METHOD ReadPropertyStatusFlags : HRESULT
VAR_INPUT
	stateFlags : REFERENCE TO ST_BA_StatusFlags;
END_VAR
VAR
	_flags : DWORD;
	_size : DINT := 2;
END_VAR
IF (ipObj <> 0) AND (__ISVALIDREF(stateFlags)) THEN
	ReadPropertyStatusFlags:=ReadProperty(E_BACnetPropIdentifier.PropStatusFlags, ADR(_flags), ADR(_size));
	
	IF (ReadPropertyStatusFlags = S_OK) THEN
		stateFlags.bInAlarm:= F_BACnet_IsBitFieldBitSet(_flags, E_BACnet_StatusFlags.eInAlarm);
		stateFlags.bFault:= F_BACnet_IsBitFieldBitSet(_flags, E_BACnet_StatusFlags.eFault);
		stateFlags.bOverridden:= F_BACnet_IsBitFieldBitSet(_flags, E_BACnet_StatusFlags.eOverridden);
		stateFlags.bOutOfService:= F_BACnet_IsBitFieldBitSet(_flags, E_BACnet_StatusFlags.eOutOfService);
	END_IF
ELSE
	ReadPropertyStatusFlags := E_FAIL;
END_IF
END_METHOD

METHOD ReadPropertyString : HRESULT
VAR_INPUT
	ePropID : E_BACnetPropIdentifier;
	value : REFERENCE TO T_MaxString;
END_VAR
VAR
	_size : UDINT := 255;
	_fbDecode : FB_BACnet_StringExtDecode;
END_VAR
IF (ipObj <> 0) AND (__ISVALIDREF(value)) THEN
	_size:=SIZEOF(BACnet_Globals.stADSBuffer);
	ReadPropertyString:=ReadProperty(ePropID, ADR(BACnet_Globals.stADSBuffer), ADR(_size));
	
	IF (ReadPropertyString = S_OK) THEN
		memset(ADR(value)+_size,0,1);
		_fbDecode(pChrStringExt:=ADR(BACnet_Globals.stADSBuffer), pOutString:=ADR(value), nOutSize:=_size);
		
		IF NOT _fbDecode.bValid THEN
			ReadPropertyString := E_FAIL;	
		END_IF
	END_IF
ELSE
	ReadPropertyString := E_FAIL;
END_IF
END_METHOD

METHOD ReadPropertyUDInt : HRESULT
VAR_INPUT
	ePropID : E_BACnetPropIdentifier;
	value : REFERENCE TO UDINT;
END_VAR
VAR
	_size : DINT := 4;
END_VAR
IF (ipObj <> 0) AND (__ISVALIDREF(value)) THEN
	ReadPropertyUDInt := ReadProperty(ePropID, ADR(value), ADR(_size));
ELSE
	ReadPropertyUDInt := E_FAIL;
END_IF
END_METHOD

METHOD ReadPropertyUnit : HRESULT
VAR CONSTANT
	ePropID : E_BACnetPropIdentifier := E_BACnetPropIdentifier.PropUnits;
END_VAR
VAR_INPUT
	value : REFERENCE TO E_BA_Unit;
END_VAR
VAR
	_size : DINT := 4;
END_VAR
IF (ipObj <> 0) AND (__ISVALIDREF(value)) THEN
	ReadPropertyUnit := ReadProperty(ePropID, ADR(value), ADR(_size));
ELSE
	ReadPropertyUnit := E_FAIL;
END_IF
END_METHOD

METHOD ReadPropertyWeeklySched : HRESULT
VAR_IN_OUT
	aWeek							: ARRAY[*, *] OF ST_BA_SchedEntry;
END_VAR
VAR_INPUT
	eDatatype						: E_BACnet_ValueChoice;
END_VAR
VAR			
	// General:
	nLenTmp							: UDINT;
	nLength							: DINT;
	
	_cbTmpSize						: UDINT;
	_cbTotalEntry					: UDINT;
	_cbTotalBuf						: UDINT;
	
	// Scheduler:
	_pDailySched					: POINTER TO ST_BACnet_DailySchedule;
	_pTimeValue						: POINTER TO ST_BACnet_TimeValueList;
	_pOldTimeValue					: POINTER TO ST_BACnet_TimeValueList;
	_nDayTmp						: DINT;
	_nDayEntryTmp					: DINT;
	_nDays							: UINT;
END_VAR
IF (ipObj = 0) THEN
	_hResult := E_FAIL;
	
ELSIF (eDataType = E_BACnet_ValueChoice.eNullValue) THEN
	iOwner.LogMsg.Show(ADSLOG_MSGTYPE_ERROR, 'RWS05', 'Invalid datatype!', TRUE);
	_hResult := E_FAIL;
ELSE
	nLength := SIZEOF(BACnet_Globals.aDefaultBuffer);
	_hResult := ReadProperty(E_BACnetPropIdentifier.PropWeeklySchedule, ADR(BACnet_Globals.aDefaultBuffer), ADR(nLength));
	
	IF (SUCCEEDED(_hResult)) THEN
		IF (nLength > 0) THEN
			// Clear content:
			_nDayTmp := F_BA_WeeklySchedSize(aWeek);
			MEMSET(aWeek, 0, TO_UDINT(F_BA_WeeklySchedSize(aWeek)));
			
			// Point to first data:
			_pDailySched := ADR(BACnet_Globals.aDefaultBuffer);
			_pTimeValue := ADR(_pDailySched^.stListEntry);
			_nDayEntryTmp := LOWER_BOUND(aWeek, 2);
			_nDayTmp := LOWER_BOUND(aWeek, 1);
			
			WHILE (_pTimeValue <> 0) AND SUCCEEDED(_hResult) DO
				(* check entry size of time value *)
				IF (_pTimeValue^.nEntrySize AND 16#7FFFFFFF) > 0 THEN
					(* check internal schedule buffer index *)
					IF (_nDayTmp > E_BA_Weekday.eSunday) THEN
						iOwner.LogMsg.Show(ADSLOG_MSGTYPE_ERROR, 'RWS23', 'Wrong day index!', TRUE);
						_hResult := E_FAIL;
					ELSE
						IF (_nDayEntryTmp <= TO_INT(BACnet_Globals.nDataField_MaxDayEntry)) THEN
							Sched_ReadEntry(eDatatype, _pTimeValue, ADR(aWeek[_nDayTmp, _nDayEntryTmp]));							
							_nDayEntryTmp := _nDayEntryTmp + 1;
						ELSE
							iOwner.LogMsg.Show(ADSLOG_MSGTYPE_WARN, 'RWS74', 'Max. count of entries reached!', TRUE);
						END_IF
	
						(* next time value entry *)
						(* check if next time value entry available *)
						IF (NOT Sched_SetNextTimeVal(_pDailySched, _pTimeValue, _cbTmpSize, _pOldTimeValue)) THEN
							(* update pointer each cycle (even if no day follows!) *)
							(* check for next day *)
							IF (NOT Sched_SetNextDay(_pDailySched, _cbTmpSize, _cbTotalBuf, _pOldTimeValue, _nDayTmp, _nDayEntryTmp, _pTimeValue)) THEN
								// Job done!
								EXIT;
							END_IF
						END_IF
					END_IF
	
				ELSE
					(* update pointer each cycle (even if no day follows!) *)
					(* No timevalue entry, check if next day element exists and pointer is plausible *)
					IF (Sched_SetNextDay(_pDailySched, _cbTmpSize, _cbTotalBuf, _pOldTimeValue, _nDayTmp, _nDayEntryTmp, _pTimeValue)) THEN
						
						// Check pointer:
						IF (_pDailySched + (_pDailySched^.nEntrySize AND 16#7FFFFFFF)) >= (ADR(BACnet_Globals.aDefaultBuffer) + SIZEOF(BACnet_Globals.aDefaultBuffer)) THEN
							iOwner.LogMsg.Show(ADSLOG_MSGTYPE_ERROR, 'RWS96', 'Insufficient buffer size!', TRUE);
							_hResult := E_FAIL;
						END_IF
					ELSE
						// Job done!
						EXIT;
					END_IF
				END_IF
				
				// Check bounds:
				IF (_nDayTmp > UPPER_BOUND(aWeek, 1)) OR (_nDayEntryTmp > UPPER_BOUND(aWeek, 2)) THEN
					EXIT;
				END_IF
			END_WHILE
		END_IF
	END_IF
END_IF

ReadPropertyWeeklySched := _hResult;
END_METHOD

METHOD INTERNAL GetSyncHandleMode : BOOL
VAR_INPUT
	eMode		: E_BA_FullSyncMode;
END_VAR
VAR_OUTPUT
	eResult		: E_BA_SyncMode;
END_VAR
CASE (eMode) OF
	eSync_FromSupplement:
		eResult := E_BA_SyncMode.eFromSupplement;
		
	eSync_ToSupplement,
	eFullSync_InitSupplement,
	eFullSync_InitPLC:
		eResult := E_BA_SyncMode.eToSupplement;
ELSE
	eResult := E_BA_SyncMode.eNone;
END_CASE

GetSyncHandleMode := (eResult <> E_BA_SyncMode.eNone);
END_METHOD

METHOD PRIVATE AddListElement : BOOL
VAR_INPUT
	ePropID				: E_BACnetPropIdentifier;
	nIndex				: DINT;
	nSize				: DINT;
	pValue				: PVOID;
END_VAR
VAR
	nListLen			: DINT;
	_size				: DINT := SIZEOF(DINT);
END_VAR
// Read current element count:
IF ipObj.SyncReadProperty(ePropID, ADR(nListLen), ADR(_size), 0) = S_OK THEN
	IF nListLen < nIndex THEN
		// Add new element to list:
		AddListElement := (ipObj.SyncWriteProperty(ePropID, pValue, nSize, 16#FFFFFFFE) = S_OK);
	ELSE
		AddListElement := TRUE;
	END_IF
END_IF
END_METHOD

METHOD PRIVATE ApplySyncHandler : BOOL
VAR
	_i		: E_BA_SyncMode;
END_VAR
ApplySyncHandler := TRUE;

// Apply requested sync handlers:
FOR _i := E_BA_SyncMode.eFromSupplement TO E_BA_SyncMode.eToSupplement DO
	IF (aReqSyncHandlers[_i] > 0) THEN
		IF (NOT SetPropertyCount(aReqSyncHandlers[_i], _i)) THEN
			ApplySyncHandler := FALSE;
		END_IF
	END_IF
END_FOR
END_METHOD

METHOD PRIVATE EvaluatePropSync
VAR_INPUT
	hResult		: HRESULT;
	eSyncMode	: E_BA_FullSyncMode;
	bCyclic		: BOOL := FALSE;
END_VAR
VAR
	_eMode		: E_BA_SyncMode	:= E_BA_SyncMode.eNone;
END_VAR
IF (SUCCEEDED(hResult)) THEN
	// Cyclic property synchronization:
	IF ((bCyclic) AND (eSyncMode > eSync_FromSupplement)) THEN
		nCycPropCnt := (nCycPropCnt+1);
	END_IF
	
	// Increment SyncHandlers:
	IF (GetSyncHandleMode(eSyncMode, eResult=>_eMode)) THEN
		aSyncHandlers[_eMode] := (aSyncHandlers[_eMode]+1);
	END_IF
END_IF
END_METHOD

METHOD RequestSyncHandlers : BOOL
VAR_INPUT
	nFromSupplement		: UDINT		:= 0;
	nToSupplement		: UDINT		:= 0;
END_VAR
aReqSyncHandlers[E_BA_SyncMode.eFromSupplement] := (aReqSyncHandlers[E_BA_SyncMode.eFromSupplement]+nFromSupplement);
aReqSyncHandlers[E_BA_SyncMode.eToSupplement] := (aReqSyncHandlers[E_BA_SyncMode.eToSupplement]+nToSupplement);
END_METHOD

METHOD RequestSyncHandlersEx : BOOL
VAR_INPUT
	eMode		: E_BA_FullSyncMode;
	nCount		: UDINT		:= 0;
END_VAR
VAR
	_eMode		: E_BA_SyncMode	:= E_BA_SyncMode.eNone;
END_VAR
IF (GetSyncHandleMode(eMode, eResult=>_eMode)) THEN
	aReqSyncHandlers[_eMode] := (aReqSyncHandlers[_eMode]+nCount);
	
	RequestSyncHandlersEx := TRUE;
END_IF
END_METHOD

METHOD SyncProperty : HRESULT
VAR_INPUT
	ePropID : E_BACnetPropIdentifier;
	nSize : UDINT;
	pValue : PVOID;
	bCOVTrig : POINTER TO BOOL := 0;
	eSyncMode : E_BA_FullSyncMode;
	bCyclic : BOOL := FALSE;
END_VAR
VAR
	nIndex : UDINT := 16#FFFFFFFF;
	_bCOV		: POINTER TO BYTE;
END_VAR
IF (ipObj <> 0) THEN
	SyncProperty := SEL(Error, ipObj.SyncPropertyData(ePropID, nSize, pValue, bCOVTrig, 0, nIndex, TO_UINT(eSyncMode)), E_FAIL);
	EvaluatePropSync(SyncProperty, eSyncMode, bCyclic);
	
	IF (SUCCEEDED(SyncProperty)) AND_THEN (bCOVTrig <> 0) THEN
		// Initialize COV indication:
		bCOVTrig^ := FALSE;
	END_IF
	
				
END_IF
END_METHOD

METHOD SyncPropertyCOV : BOOL
VAR_INPUT
	ePropertyID : E_BACnetPropIdentifier;
	bCOVTrig : POINTER TO BOOL;
END_VAR
VAR
	_hResult : HRESULT;
END_VAR
IF (ipObj <> 0) AND_THEN (bCOVTrig <> 0) THEN
	// Initialize COV indication:
	_hResult := SyncProperty(ePropertyID, 0, 0, bCOVTrig, eSync_FromSupplement, FALSE);
	IF (_hResult <> S_OK) THEN
		iOwner.LogMsg.Show2(ADSLOG_MSGTYPE_ERROR, 'SPCOV03', 'Initialize COV-Trigger of property "%d" failed (Error: 0x%x)!', F_INT(ePropertyID), F_DINT(_hResult), TRUE);
	ELSE
		// Initialize COV indication:
		bCOVTrig^ := FALSE;
		
		SyncPropertyCOV := TRUE;
	END_IF
END_IF
END_METHOD

METHOD SyncPropertyIdx : HRESULT
VAR_INPUT
	ePropID : E_BACnetPropIdentifier;
	nSize : UDINT;
	pValue : PVOID;
	nIndex : INT := -1;
	pData : PVOID := 0;
	eSyncMode : E_BA_FullSyncMode;
	bCyclic : BOOL := FALSE;
END_VAR
IF (ipObj <> 0) THEN
	SyncPropertyIdx := SEL(Error, ipObj.SyncPropertyData(ePropID, nSize, pValue, pData, 0, TO_UDINT(nIndex), TO_UINT(eSyncMode)), E_FAIL);
	EvaluatePropSync(_hResult, eSyncMode, bCyclic);
END_IF
END_METHOD

METHOD SyncPropertyList : BOOL
VAR_INPUT
	ePropID				: E_BACnetPropIdentifier;
	pList				: PVOID;
	nItemSize			: UDINT;
	nItemCount			: UDINT;
	eSyncMode			: E_BA_FullSyncMode;
	bValidate			: BOOL						:= FALSE;			// Check items contents and stops synchronization if an used items is found.
END_VAR
VAR
	_nTemp				: UDINT;
	_pValue				: PVOID;
END_VAR
IF (bValidate) THEN
	RemoveListElements(ePropID);
END_IF

IF (ipObj <> 0) AND_THEN (pList <> 0) AND (nItemSize > 0) AND (nItemCount > 0) THEN
	FOR _nTemp := 1 TO nItemCount DO
		_pValue := (pList + ((_nTemp-1) * nItemSize));
		
		IF (bValidate) AND_THEN (F_BA_ByteCmp(_pValue, nItemSize, 0) = 0) THEN
			// Synchronization of used items completed:
			EXIT;
		END_IF
	
		IF NOT AddListElement(ePropID, TO_DINT(_nTemp), SIZEOF(STRING), _pValue) THEN
			RETURN;
		ELSIF SyncPropertyIdx(ePropID, SIZEOF(STRING), _pValue, TO_INT(_nTemp), 0, eSyncMode, FALSE) <> S_OK THEN
			RETURN;
		END_IF
	END_FOR
	
	SyncPropertyList := TRUE;
END_IF
END_METHOD

METHOD SyncPropertyPvPrio : HRESULT
VAR_INPUT
	ePropID : E_BACnetPropIdentifier;
	nSize : UDINT;
	pValue : PVOID;
	bEnPriority : POINTER TO BOOL;
	ePriority : E_BACnet_Priority;
	pData : PVOID := 0;
	eSyncMode : E_BA_FullSyncMode;
	bCyclic : BOOL := FALSE;
END_VAR
IF (ipObj <> 0) THEN
	SyncPropertyPvPrio := SEL(Error, ipObj.SyncPropertyData(ePropID, nSize, pValue, pData, bEnPriority, TO_UDINT(ePriority), TO_UINT(eSyncMode)), E_FAIL);
	EvaluatePropSync(_hResult, eSyncMode, bCyclic);
END_IF
END_METHOD

METHOD WriteProperty : HRESULT
VAR_INPUT
	ePropID : E_BACnetPropIdentifier;
	pData : PVOID;
	nData : DINT;
END_VAR
IF (ipObj <> 0) THEN
	WriteProperty:=ipObj.SyncWriteProperty(TO_INT(ePropID), pData, nData, 16#FFFFFFFF);
	
	IF (WriteProperty <> S_OK) THEN
		iOwner.LogMsg.Show2(ADSLOG_MSGTYPE_ERROR, 'WP5', 'Writing property "%d" failed (Error "0x%x")!', F_INT(ePropID), F_DINT(WriteProperty), TRUE);
	END_IF
ELSE
	WriteProperty := E_FAIL;
END_IF
END_METHOD

METHOD WritePropertyBool : HRESULT
VAR_INPUT
	ePropID : E_BACnetPropIdentifier;
	bValue : BOOL;
END_VAR
IF (ipObj <> 0) THEN
	WritePropertyBool := WriteProperty(ePropID, ADR(bValue), SIZEOF(bValue));
ELSE
	WritePropertyBool := E_FAIL;
END_IF
END_METHOD

METHOD WritePropertyDateList : HRESULT
VAR_IN_OUT
	aDateList				: ARRAY[*] OF ST_BA_CalendarEntry;
END_VAR
VAR
	_i						: DINT;
	
	_stEntry				: POINTER TO ST_BACnet_CalendarEntry;
	_cbTotalBuf				: UDINT;
END_VAR
IF (ipObj = 0) THEN
	_hResult := E_FAIL;
ELSE
	_stEntry := ADR(BACnet_Globals.aDefaultBuffer);
	_cbTotalBuf := 0;
	
	FOR _i := LOWER_BOUND(aDateList, 1) TO UPPER_BOUND(aDateList, 1) DO
		IF (F_BACnet_ToDateListEntry(ADR(aDateList[_i]), stResult=>_stEntry^)) THEN		
			_stEntry := (_stEntry+SIZEOF(ST_BACnet_CalendarEntry));
			_cbTotalBuf := (_cbTotalBuf+SIZEOF(ST_BACnet_CalendarEntry));
		END_IF
	END_FOR
	
	// Write data:
	_hResult := WriteProperty(E_BACnetPropIdentifier.PropDateList, ADR(BACnet_Globals.aDefaultBuffer), TO_DINT(_cbTotalBuf));
END_IF	

WritePropertyDateList := _hResult;
END_METHOD

METHOD WritePropertyEventEnable : HRESULT
VAR_INPUT
	bToNormal : BOOL;
	bToFault : BOOL;
	bToOffNormal : BOOL;
END_VAR
VAR
	_flags : WORD := 16#0005;
END_VAR
IF (ipObj <> 0) THEN
	IF bToNormal THEN
		_flags:=_flags OR 16#2000;
	END_IF
	IF bToFault THEN
		_flags:=_flags OR 16#4000;
	END_IF
	IF bToOffNormal THEN
		_flags:=_flags OR 16#8000;
	END_IF

	WritePropertyEventEnable := WriteProperty(E_BACnetPropIdentifier.PropEventEnable, ADR(_flags), 2);
ELSE
	WritePropertyEventEnable := E_FAIL;
END_IF
END_METHOD

METHOD WritePropertyEventParameter : HRESULT
VAR_IN_OUT
	stEventParameter		: ST_BACnet_EventParameter;
END_VAR
VAR
	_cbTotalBuf				: UDINT;
END_VAR
IF (ipObj = 0) THEN
	_hResult := E_FAIL;
ELSE
	CASE stEventParameter.eEventType OF
		E_BACnet_EventType.eOutOfRange:
			stEventParameter.nArgSize := SIZEOF(ST_BACnet_EventOutOfRange);
		E_BACnet_EventType.eUnsignedRange:
			stEventParameter.nArgSize := SIZEOF(ST_BACnet_EventUnsignedRange);
		ELSE
			IF stEventParameter.nArgSize = 0 THEN
				WritePropertyEventParameter := E_FAIL;
				RETURN;
			END_IF
	END_CASE
	_cbTotalBuf := TO_UDINT(8 + stEventParameter.nArgSize);
	_hResult := WriteProperty(E_BACnetPropIdentifier.PropEventParameters, ADR(stEventParameter), TO_DINT(_cbTotalBuf));
END_IF	

WritePropertyEventParameter := _hResult;
END_METHOD

METHOD WritePropertyExceptionSched : HRESULT
VAR_IN_OUT
	aCalendar			: ARRAY[*] OF ST_BACnet_SchedCalendar;
	aException			: ARRAY[*] OF ST_BACnet_SchedException;
END_VAR
VAR_INPUT
	eDatatype			: E_BACnet_ValueChoice;
END_VAR
VAR
	_nEntry				: DINT;
	_nSchedEntry		: INT;
	_hResult			: HRESULT;
	_pDailySched		: POINTER TO ST_BACnet_SpecialEventList;
	_pDailySchedOld		: POINTER TO ST_BACnet_SpecialEventList;
	_cbTotalSize		: UDINT;
	_cbTmpSize			: UDINT;
	_calObjId 			: T_BACnet_ObjectIdentifier;
	_pTimeValue			: POINTER TO ST_BACnet_TimeValueList;
	_pOldTimeValue		: POINTER TO ST_BACnet_TimeValueList;
	
	// [Bug-Workaround]: Diese scheiss Firma 3S
	// CASE (aCalendar[_nEntry].aEntry[_nSchedEntry].eState) OF			// "...aEntry[_nTimeValue]" ist immer der Pointer auf "aEntry[1]" :(
	_pCalEntry			: POINTER TO ST_BA_SchedEntry;
	
	// [Bug-Workaround]: Diese scheiss Firma 3S
	// Sched_ReadEntry(eDatatype, _pTimeValue, aException[_nExcEntry].aEntry[_nTimeValue]);			// "...aEntry[_nTimeValue]" ist immer der Pointer auf "aEntry[1]" :(
	_pExceptEntry		: POINTER TO ST_BA_SchedEntry;
END_VAR
IF ipObj = 0 THEN
	_hResult := E_FAIL;
ELSE
	_pDailySched := ADR(BACnet_Globals.aDefaultBuffer);
	_pDailySchedOld := 0;
	_cbTotalSize := 0;
	
	FOR _nEntry := LOWER_BOUND(aCalendar, 1) TO UPPER_BOUND(aCalendar, 1) DO
		IF F_BACnet_IsObjIdentifierValid(aCalendar[_nEntry].tRefCalendarID) THEN
			MEMSET(ADR(_pDailySched^.stEvent), 0, SIZEOF(_pDailySched^.stEvent));
			_pDailySched^.nEntrySize := SIZEOF(_pDailySched^.stEvent);
			_pDailySched^.nRes := 0;
			_pDailySched^.stEvent.eEventChoice := E_BACnet_SpecialEventChoice.eCalendarReference;
			_pDailySched^.stEvent.nEventPriority := SEL(F_BACnet_IsPriorityValid(aCalendar[_nEntry].eEventPriority), 1, TO_UDINT(aCalendar[_nEntry].eEventPriority));
				
			IF  _pDailySchedOld <> 0 THEN
				_pDailySchedOld^.nEntrySize := _pDailySchedOld^.nEntrySize + 16#80000000;
			END_IF
			
			_calObjId := aCalendar[_nEntry].tRefCalendarID;
			MEMCPY(ADR(_pDailySched^.stEvent.eCalEntryChoice), ADR(_calObjId), SIZEOF(_calObjId));
			
			_pOldTimeValue := 0;
			_pTimeValue:= F_BACnet_EndOf(_pDailySched, SIZEOF(ST_BACnet_SpecialEventList));
			_pCalEntry := ADR(aCalendar[_nEntry].aEntry[1]);
			FOR _nSchedEntry:=1 TO BACnet_Param.nSched_EntryCount DO
				CASE (_pCalEntry^.eState) OF
					E_BA_SchedEntryState.eNull,
					E_BA_SchedEntryState.eValue:
						 _pTimeValue^.nEntrySize := 0;
						 _pTimeValue^.nRes := 0;
						 
						 // Set flag "next entry" to the previous element:
						IF (_nSchedEntry > 1) AND (_pOldTimeValue <> 0) THEN
							_pOldTimeValue^.nEntrySize := _pOldTimeValue^.nEntrySize + 16#80000000;
						END_IF
						
						Sched_WriteEntry(eDatatype, _pTimeValue, _pCalEntry); 
						
						_pDailySched^.nEntrySize := _pDailySched^.nEntrySize + F_BACnet_AlignedSize(_pTimeValue^.nEntrySize) + SIZEOF(_pTimeValue^.nEntrySize) + SIZEOF(_pTimeValue^.nRes);	
											
						_pOldTimeValue := _pTimeValue;
						_pTimeValue := _pTimeValue +  F_BACnet_AlignedSize(_pTimeValue^.nEntrySize AND 16#7FFFFFFF) + SIZEOF(_pTimeValue^.nEntrySize) + SIZEOF(_pTimeValue^.nRes);					 
				END_CASE
				_pCalEntry := (_pCalEntry+SIZEOF(ST_BA_SchedEntry));
			END_FOR
			IF _pOldTimeValue = 0 THEN // no TimeValue entry -> empty list
				_pDailySched^.nEntrySize := _pDailySched^.nEntrySize + SIZEOF(_pTimeValue^.nEntrySize) + SIZEOF(_pTimeValue^.nRes);
				_pTimeValue^.nEntrySize := 0;
				_pTimeValue^.nRes := 0;
			END_IF
		
			_cbTotalSize := _cbTotalSize + F_BACnet_AlignedSize(_pDailySched^.nEntrySize AND 16#7FFFFFFF) + SIZEOF(_pDailySched^.nEntrySize) + SIZEOF(_pDailySched^.nRes);	
			_pDailySchedOld := _pDailySched;
			_pDailySched := _pDailySched +  F_BACnet_AlignedSize(_pDailySched^.nEntrySize AND 16#7FFFFFFF) + SIZEOF(_pDailySched^.nEntrySize) + SIZEOF(_pDailySched^.nRes);					 		
		END_IF
	END_FOR
	
	FOR _nEntry := LOWER_BOUND(aException, 1) TO UPPER_BOUND(aException, 1) DO
		IF aException[_nEntry].eType <> E_BA_DateValChoice.Invalid THEN
			MEMSET(ADR(_pDailySched^.stEvent), 0, SIZEOF(_pDailySched^.stEvent));
			_pDailySched^.nEntrySize := SIZEOF(_pDailySched^.stEvent);
			_pDailySched^.nRes := 0;
			_pDailySched^.stEvent.eEventChoice := E_BACnet_SpecialEventChoice.eCalendarEntry;
			IF aException[_nEntry].nEventPriority > 0 AND aException[_nEntry].nEventPriority < 17 THEN
				_pDailySched^.stEvent.nEventPriority := aException[_nEntry].nEventPriority; 
			ELSE
				_pDailySched^.stEvent.nEventPriority := 1;
			END_IF
			IF _pDailySchedOld <> 0 THEN
				_pDailySchedOld^.nEntrySize := _pDailySchedOld^.nEntrySize + 16#80000000;
			END_IF
			
			_pDailySched^.stEvent.eCalEntryChoice := aException[_nEntry].eType-1;
			_pDailySched^.stEvent.uCalEntry := aException[_nEntry].uDate;
			
			_pOldTimeValue := 0;
			_pTimeValue:= F_BACnet_EndOf(_pDailySched, SIZEOF(ST_BACnet_SpecialEventList));
			_pExceptEntry := ADR(aException[_nEntry].aEntry[1]);
			FOR _nSchedEntry:=1 TO BACnet_Param.nSched_EntryCount DO
				CASE (_pExceptEntry^.eState) OF
					E_BA_SchedEntryState.eNull,
					E_BA_SchedEntryState.eValue:
						 _pTimeValue^.nEntrySize := 0;
						 _pTimeValue^.nRes := 0;
						 
						 // Set flag "next entry" to the previous element:
						IF (_nSchedEntry > 1) AND (_pOldTimeValue <> 0) THEN
							_pOldTimeValue^.nEntrySize := _pOldTimeValue^.nEntrySize + 16#80000000;
						END_IF
						
						Sched_WriteEntry(eDatatype, _pTimeValue, _pExceptEntry); 
						
						_pDailySched^.nEntrySize := _pDailySched^.nEntrySize + F_BACnet_AlignedSize(_pTimeValue^.nEntrySize) + SIZEOF(_pTimeValue^.nEntrySize) + SIZEOF(_pTimeValue^.nRes);	
											
						_pOldTimeValue := _pTimeValue;
						_pTimeValue := _pTimeValue +  F_BACnet_AlignedSize(_pTimeValue^.nEntrySize AND 16#7FFFFFFF) + SIZEOF(_pTimeValue^.nEntrySize) + SIZEOF(_pTimeValue^.nRes);					 
				END_CASE
				_pExceptEntry := (_pExceptEntry+SIZEOF(ST_BA_SchedEntry));
			END_FOR
			IF _pOldTimeValue = 0 THEN // no TimeValue entry -> empty list
				_pDailySched^.nEntrySize := _pDailySched^.nEntrySize + SIZEOF(_pTimeValue^.nEntrySize) + SIZEOF(_pTimeValue^.nRes);
				_pTimeValue^.nEntrySize := 0;
				_pTimeValue^.nRes := 0;
			END_IF
						
			_cbTotalSize := _cbTotalSize + F_BACnet_AlignedSize(_pDailySched^.nEntrySize AND 16#7FFFFFFF) + SIZEOF(_pDailySched^.nEntrySize) + SIZEOF(_pDailySched^.nRes);	
			_pDailySchedOld := _pDailySched;
			_pDailySched := _pDailySched +  F_BACnet_AlignedSize(_pDailySched^.nEntrySize AND 16#7FFFFFFF) + SIZEOF(_pDailySched^.nEntrySize) + SIZEOF(_pDailySched^.nRes);					 
		END_IF
	END_FOR
	
	IF (_cbTotalSize = 0) THEN
		// Indicate empty exception property:
		_cbTotalSize := 8;
		MEMSET(ADR(BACnet_Globals.aDefaultBuffer), 0, _cbTotalSize);
	END_IF
	
	// Write data:
	_hResult := WriteProperty(E_BACnetPropIdentifier.PropExceptionSchedule, ADR(BACnet_Globals.aDefaultBuffer), TO_DINT(_cbTotalSize));
END_IF

IF (F_BACnet_FilterErrCode(_hResult) = TO_DINT(E_AdsErr.DEVICE_ACCESSDENIED)) THEN
	// Fallback to old (valid) property value:
	ReadPropertyExceptionSched(aCalendar, aException, eDataType);
END_IF

WritePropertyExceptionSched := _hResult;
END_METHOD

METHOD WritePropertyLimitEnable : HRESULT
VAR_INPUT
	bLowLimitEnable : BOOL;
	bHighLimitEnable : BOOL;
END_VAR
VAR
	_flags : WORD := 16#0006;
END_VAR
IF (ipObj <> 0) THEN
	IF bLowLimitEnable THEN
		_flags:=_flags OR 16#8000;
	END_IF
	IF bHighLimitEnable THEN
		_flags:=_flags OR 16#4000;
	END_IF

	WritePropertyLimitEnable := WriteProperty(E_BACnetPropIdentifier.PropLimitEnable, ADR(_flags), 2);
ELSE
	WritePropertyLimitEnable := E_FAIL;
END_IF
END_METHOD

METHOD WritePropertyLogBuffer : HRESULT
VAR_IN_OUT
	aLogBuffer						: ARRAY [*] OF ST_BA_TrendEntry;
END_VAR
IF (ipObj = 0) THEN
	_hResult := E_FAIL;
ELSE
	_hResult := S_OK;
	// ...
	
END_IF	

WritePropertyLogBuffer := _hResult;
END_METHOD

METHOD WritePropertyNotifyType : HRESULT
VAR CONSTANT
	ePropID : E_BACnetPropIdentifier := E_BACnetPropIdentifier.PropNotifyType;
END_VAR
VAR_INPUT
	value : E_BACnet_NotifyType;
END_VAR
IF (ipObj <> 0) THEN
	WritePropertyNotifyType := WriteProperty(ePropID, ADR(value), SIZEOF(value));
ELSE
	WritePropertyNotifyType := E_FAIL;
END_IF
END_METHOD

METHOD WritePropertyNull : HRESULT
VAR_INPUT
	ePropID : E_BACnetPropIdentifier;
	prio : BYTE := 0;
END_VAR
IF (ipObj <> 0) THEN
	WritePropertyNull := ipObj.SyncWriteProperty(TO_INT(ePropID), 0, 0, prio);
	
	IF (WritePropertyNull <> S_OK) THEN
		F_BA_LogMessage2(ADSLOG_MSGTYPE_ERROR, 'WPN5', 'Writing property "%d" failed (Error "0x%x")!', F_INT(ePropID), F_DINT(WritePropertyNull));
	END_IF
ELSE
	WritePropertyNull := E_FAIL;
END_IF
END_METHOD

METHOD WritePropertyReal : HRESULT
VAR_INPUT
	ePropID : E_BACnetPropIdentifier;
	fValue : REAL;
END_VAR
IF (ipObj <> 0) THEN
	WritePropertyReal := WriteProperty(ePropID, ADR(fValue), SIZEOF(fValue));
ELSE
	WritePropertyReal := E_FAIL;
END_IF
END_METHOD

METHOD WritePropertyRealPrio : HRESULT
VAR_INPUT
	ePropID : E_BACnetPropIdentifier;
	fValue : REAL;
	prio : BYTE := 0;
END_VAR
IF (ipObj <> 0) THEN
	WritePropertyRealPrio := ipObj.SyncWriteProperty(TO_INT(ePropID), ADR(fValue), SIZEOF(fValue), prio);
	
	IF (WritePropertyRealPrio <> S_OK) THEN
		F_BA_LogMessage2(ADSLOG_MSGTYPE_ERROR, 'WPRP5', 'Writing property "%d" failed (Error "0x%x")!', F_INT(ePropID), F_DINT(WritePropertyRealPrio));
	END_IF
ELSE
	WritePropertyRealPrio := E_FAIL;
END_IF
END_METHOD

METHOD WritePropertyRecipientList : HRESULT
VAR_IN_OUT
	aRecipientList			: ARRAY[*] OF ST_BACnet_Destination;
END_VAR
// [Bugworkaround]
// > _stUnused" has to be static, otherwise its memory can be initialized incorrectly by PLC :(
VAR_STAT
	_nLowerBound			: DINT;
	_nCount					: DINT;
	_stUnused				: ST_BACnet_Destination;
END_VAR
_hResult := E_FAIL;

IF (ipObj <> 0) THEN
	_nLowerBound := LOWER_BOUND(aRecipientList, 1);
	_nCount := F_BA_GetUsedEntryCount(aRecipientList, _nLowerBound, UPPER_BOUND(aRecipientList, 1), _stUnused);
	
	IF (_nCount > 0) THEN
		_hResult := WriteProperty(E_BACnetPropIdentifier.PropRecipientList, aRecipientList, SIZEOF(ST_BACnet_Destination) * (_nLowerBound + _nCount - 1));
	ELSE
		IF RemoveArrayElements(E_BACnetPropIdentifier.PropRecipientList) THEN
			_hResult := S_OK;
		END_IF
	END_IF
END_IF

IF (F_BACnet_FilterErrCode(_hResult) = TO_DINT(E_AdsErr.DEVICE_ACCESSDENIED)) THEN
	// Fallback to old (valid) property value:
	ReadPropertyRecipientList(aRecipientList);
END_IF

WritePropertyRecipientList := _hResult;
END_METHOD

METHOD WritePropertyReference : HRESULT
VAR_INPUT
	eProperty			: E_BACnetPropIdentifier;
END_VAR
VAR_IN_OUT
	stReference			: ST_BACnet_ObjectPropertyReference;
END_VAR
VAR
	_pEntry				: ST_BACnet_DeviceObjectPropertyReference;
END_VAR
IF (ipObj <> 0) THEN
	IF (stReference.iObject = 0) THEN
		// Set referred object to NULL.
	ELSE
		_pEntry.stValidFields.bPropertyIdentifier := TRUE;
		_pEntry.stValidFields.bObjectId := TRUE;
		_pEntry.tObjId := stReference.iObject.ObjectID;
		_pEntry.ePropIdentifier := stReference.ePropertyId;
	END_IF
	
	WritePropertyReference := WriteProperty(eProperty, ADR(_pEntry), SIZEOF(_pEntry));
ELSE
	WritePropertyReference := E_FAIL;
END_IF
END_METHOD

METHOD WritePropertyReferenceList : HRESULT
VAR_INPUT
	eProperty			: E_BACnetPropIdentifier;
END_VAR
VAR_IN_OUT
	aReferences 		: ARRAY[*] OF ST_BACnet_ObjectPropertyReference;
END_VAR
VAR
	_pEntry				: POINTER TO ST_BACnet_DeviceObjectPropertyReference;
	_i 					: DINT;
	_nSize				: DINT;
END_VAR
IF (ipObj <> 0) THEN
	_pEntry := ADR(BACnet_Globals.aDefaultBuffer);

	FOR _i:= LOWER_BOUND(aReferences, 1) TO UPPER_BOUND(aReferences, 1) DO
		IF (aReferences[_i].iObject <> 0) THEN
			MEMSET(_pEntry, 0, SIZEOF(ST_BACnet_DeviceObjectPropertyReference));
			
			_pEntry^.stValidFields.bPropertyIdentifier := TRUE;
			_pEntry^.stValidFields.bObjectId := TRUE;
			_pEntry^.tObjId := aReferences[_i].iObject.ObjectID;
			_pEntry^.ePropIdentifier := aReferences[_i].ePropertyId;
			
			_nSize := _nSize + SIZEOF(ST_BACnet_DeviceObjectPropertyReference);
			_pEntry := F_BACnet_EndOf(_pEntry, SIZEOF(ST_BACnet_DeviceObjectPropertyReference));
		END_IF
	END_FOR
	WritePropertyReferenceList := WriteProperty(eProperty, ADR(BACnet_Globals.aDefaultBuffer),_nSize);
ELSE
	WritePropertyReferenceList := E_FAIL;
END_IF
END_METHOD

METHOD WritePropertyReferenceList1x : HRESULT
VAR_INPUT
	eProperty			: E_BACnetPropIdentifier;
END_VAR
VAR_IN_OUT
	stReference			: ST_BACnet_ObjectPropertyReference;
END_VAR
VAR
	_aRefArray 			: POINTER TO ARRAY[1 .. 1] OF ST_BACnet_ObjectPropertyReference;
END_VAR
IF (ipObj <> 0) THEN
	_aRefArray := ADR(stReference);
	WritePropertyReferenceList1x := WritePropertyReferenceList(eProperty, _aRefArray^);
ELSE
	WritePropertyReferenceList1x := E_FAIL;
END_IF
END_METHOD

METHOD WritePropertyString : HRESULT
VAR_INPUT
	ePropID : E_BACnetPropIdentifier;
	value : T_MaxString;
END_VAR
VAR
	_nResult : UDINT;
END_VAR
IF (ipObj <> 0) THEN
	IF (F_BACnet_EncodeUTF8(
		pString		:= ADR(value),
		nString	:= TO_UDINT(LEN(value)),
		pResult		:= ADR(BACnet_Globals.stADSBuffer),
		nResult	:= SIZEOF(BACnet_Globals.stADSBuffer),
		nResultLen	:= _nResult) <> 0)
			THEN
				WritePropertyString := WriteProperty(ePropID, ADR(BACnet_Globals.stADSBuffer), TO_UINT(_nResult));
	END_IF
END_IF
END_METHOD

METHOD WritePropertyStringIdx : HRESULT
VAR_INPUT
	ePropID : E_BACnetPropIdentifier;
	str : STRING;
	idx : BYTE;
END_VAR
VAR
	_nResult : UDINT;
END_VAR
IF (ipObj <> 0) THEN
	IF (F_BACnet_EncodeUTF8(
		pString		:= ADR(str),
		nString	:= TO_UDINT(LEN(str)),
		pResult		:= ADR(BACnet_Globals.stADSBuffer),
		nResult	:= SIZEOF(BACnet_Globals.stADSBuffer),
		nResultLen	:= _nResult) <> 0)
			THEN
			WritePropertyStringIdx := ipObj.SyncWriteProperty(TO_INT(ePropID), ADR(BACnet_Globals.stADSBuffer),  TO_UINT(F_BACnet_AlignedSize(_nResult)), idx);
			
			IF (WritePropertyStringIdx <> S_OK) THEN
				F_BA_LogMessage2(ADSLOG_MSGTYPE_ERROR, 'WPSI512', 'Writing property "%d" failed (Error "0x%x")!', F_INT(ePropID), F_DINT(WritePropertyStringIdx));
			END_IF
	END_IF
END_IF
END_METHOD

METHOD WritePropertyUDInt : HRESULT
VAR_INPUT
	ePropID : E_BACnetPropIdentifier;
	nValue : UDINT;
END_VAR
IF (ipObj <> 0) THEN
	WritePropertyUDInt := WriteProperty(ePropID, ADR(nValue), SIZEOF(nValue));
ELSE
	WritePropertyUDInt := E_FAIL;
END_IF
END_METHOD

METHOD WritePropertyUInt : HRESULT
VAR_INPUT
	ePropID : E_BACnetPropIdentifier;
	nValue : UINT;
END_VAR
IF (ipObj <> 0) THEN
	WritePropertyUInt := WriteProperty(ePropID, ADR(nValue), SIZEOF(nValue));
ELSE
	WritePropertyUInt := E_FAIL;
END_IF
END_METHOD

METHOD WritePropertyUnit : HRESULT
VAR CONSTANT
	ePropID : E_BACnetPropIdentifier := E_BACnetPropIdentifier.PropUnits;
END_VAR
VAR_INPUT
	eValue : E_BA_Unit;
END_VAR
IF (ipObj <> 0) THEN
	WritePropertyUnit := WriteProperty(ePropID, ADR(eValue), SIZEOF(eValue));
ELSE
	WritePropertyUnit := E_FAIL;
END_IF
END_METHOD

METHOD WritePropertyValue : HRESULT
VAR_INPUT
	eProperty : E_BACnetPropIdentifier;
	xValue : ANY;
END_VAR
VAR
	_eValueChoice : E_BACnet_ValueChoice;
END_VAR
CASE (xValue.TypeClass) OF
	__SYSTEM.TYPE_CLASS.TYPE_REAL:
		_eValueChoice := E_BACnet_ValueChoice.eRealValue;
	__SYSTEM.TYPE_CLASS.TYPE_UDINT:
		_eValueChoice := E_BACnet_ValueChoice.eUnsignedValue;
	__SYSTEM.TYPE_CLASS.TYPE_BOOL:
		_eValueChoice := E_BACnet_ValueChoice.eBoolValue;
	__SYSTEM.TYPE_CLASS.TYPE_ENUM:
		_eValueChoice := E_BACnet_ValueChoice.eEnumerationValue;
ELSE
	iOwner.LogMsg.Show1(ADSLOG_MSGTYPE_ERROR, 'WPV30', 'Unimplemented datatype! (Type class "%d")', F_DWORD(xValue.TypeClass), TRUE);
	RETURN;
END_CASE

WritePropertyValue := WritePropertyValueEx(eProperty, _eValueChoice, xValue.diSize, xValue.pValue);
END_METHOD

METHOD WritePropertyValueEx : HRESULT
VAR_INPUT
	eProperty : E_BACnetPropIdentifier;
	eValueChoice : E_BACnet_ValueChoice;
	nSize : DINT;
	pValue : PVOID;
END_VAR
VAR
	_stData : ST_BACnet_ValueList;
	_nSize : DWORD;
END_VAR
IF (bReady) AND (nSize > 0) AND (pValue <> 0) THEN
	IF (eValueChoice = E_BACnet_ValueChoice.eEnumerationValue) THEN
		_nSize := SIZEOF(ST_BACnet_ValueList);	
		_stData.nEntrySize := TO_DWORD(SIZEOF(ST_BACnet_Value));
		_stData.listEntry.eValueChoice := eValueChoice;
		_stData.listEntry.nSize := SIZEOF(ST_BACnet_EnumerationValueType);
		_stData.listEntry.stValue.choice := E_BACnet_EnumerationValueChoice.eBinaryPV;
		_stData.listEntry.stValue.enumValue := 0;
		
		MEMCPY(ADR(_stData.listEntry.stValue.enumValue), pValue, TO_UDINT(nSize)); 
	ELSE		
		_nSize := ((SIZEOF(ST_BACnet_ValueList) - SIZEOF(ST_BACnet_EnumerationValueType)) + TO_DWORD(nSize));
		
		_stData.nEntrySize := TO_DWORD((SIZEOF(ST_BACnet_Value) - SIZEOF(ST_BACnet_EnumerationValueType) + nSize));
		_stData.listEntry.eValueChoice := eValueChoice;
		_stData.listEntry.nSize := TO_DWORD(nSize);
		
		MEMCPY(ADR(_stData.listEntry.stValue), pValue, TO_UDINT(nSize)); 
	END_IF
	
	WritePropertyValueEx := WriteProperty(eProperty, ADR(_stData), TO_DINT(F_BACnet_AlignedSize(_nSize)));
				
	IF (S_OK <> WritePropertyValueEx) THEN
		iOwner.LogMsg.Show1(ADSLOG_MSGTYPE_ERROR, 'WPVE12', 'Writing value of property "%d" failed!', F_INT(eProperty), TRUE);
	END_IF
END_IF
END_METHOD

METHOD WritePropertyWeeklySched : HRESULT
VAR_IN_OUT
	aWeek					: ARRAY[*, *] OF ST_BA_SchedEntry;
END_VAR
VAR_INPUT
	eValueChoice			: E_BACnet_ValueChoice;
END_VAR
VAR
	_cbTmpSize				: UDINT;
	_cbTotalEntry			: UDINT;
	_cbTotalBuf				: UDINT;
	_pDailySched			: POINTER TO ST_BACnet_DailySchedule;
	_pTimeValue				: POINTER TO ST_BACnet_TimeValueList;
	_pOldTimeValue			: POINTER TO ST_BACnet_TimeValueList;
	_nDay					: DINT;
	_nDayEntry				: DINT;
	_nDays					: UINT;
END_VAR
IF (ipObj = 0) THEN
	_hResult := E_FAIL;
ELSE
	// Point to first data:
	_pDailySched := ADR(BACnet_Globals.aDefaultBuffer);
	_cbTotalBuf := 0;
	_nDay := LOWER_BOUND(aWeek, 1);
	_hResult := S_OK;
	
	WHILE SUCCEEDED(_hResult) DO
		// Set timevalue pointer:
		_pTimeValue := ADR(_pDailySched^.stListEntry);
		_pTimeValue^.nEntrySize := 0;
		_pTimeValue^.nRes := 0;
		_cbTotalEntry := 0;
		_pOldTimeValue := 0;
		
		FOR _nDayEntry := LOWER_BOUND(aWeek, 2) TO UPPER_BOUND(aWeek, 2) DO			
			CASE (aWeek[_nDay, _nDayEntry].eState) OF
				E_BA_SchedEntryState.eNull,
				E_BA_SchedEntryState.eValue:
					// Set flag "next entry" to the previous element:
					IF (_nDayEntry > 1) AND (_pOldTimeValue <> 0) THEN
						_pOldTimeValue^.nEntrySize := _pOldTimeValue^.nEntrySize + 16#80000000;
					END_IF
					
					Sched_WriteEntry(eValueChoice, _pTimeValue, ADR(aWeek[_nDay, _nDayEntry])); 
					
					// Update time value pointer:
					Sched_SetNextTimeVal(_pDailySched, _pTimeValue, _cbTmpSize, _pOldTimeValue);
					
					// ...and add to total entry size counter:
					_cbTotalEntry := _cbTotalEntry + _cbTmpSize;
			END_CASE
		END_FOR
		
		// Caclulate day-entry size:
		_pDailySched^.nEntrySize := MAX(_cbTotalEntry, SIZEOF(_pDailySched^.stListEntry.nEntrySize) + SIZEOF(_pDailySched^.stListEntry.nRes));
		
		// Next day?
		IF (_nDay < UPPER_BOUND(aWeek, 1)) THEN
			_pDailySched^.nEntrySize := _pDailySched^.nEntrySize + 16#80000000;
		END_IF
		
		// Update pointer each cycle (even if no day follows!):
		IF NOT Sched_SetNextDay(_pDailySched, _cbTmpSize, _cbTotalBuf, _pOldTimeValue, _nDay, _nDayEntry, _pTimeValue) THEN
			EXIT;
		END_IF
	END_WHILE
	
	// Write data:
	_hResult := WriteProperty(E_BACnetPropIdentifier.PropWeeklySchedule, ADR(BACnet_Globals.aDefaultBuffer), TO_DINT(_cbTotalBuf));
END_IF	
	
IF (F_BACnet_FilterErrCode(_hResult) = TO_DINT(E_AdsErr.DEVICE_ACCESSDENIED)) THEN
	// Fallback to old (valid) property value:
	ReadPropertyWeeklySched(aWeek, eValueChoice);
END_IF

WritePropertyWeeklySched := _hResult;
END_METHOD

END_FUNCTION_BLOCK

// POUs/Helper/F_BACnet_GetObjId
FUNCTION F_BACnet_GetObjId : T_BACnet_ObjectIdentifier
VAR_INPUT
	eObjectType		: E_BACnetObjType;
	nObjectInstance	: UDINT;
END_VAR
VAR
END_VAR

F_BACnet_GetObjId := F_BACnet_GetObjInstance(nObjectInstance) + SHL(INT_TO_UDINT(eObjectType), 22);

END_FUNCTION

// POUs/Helper/F_BACnet_GetObjInstance
FUNCTION F_BACnet_GetObjInstance : UDINT
VAR_INPUT
	nObjectId : DWORD;
END_VAR
VAR
END_VAR

F_BACnet_GetObjInstance := nObjectId AND BACnet_Globals.nBACnetInstId_Auto;

END_FUNCTION

// POUs/Helper/F_BACnet_GetObjType
FUNCTION F_BACnet_GetObjType : E_BACnetObjType
VAR_INPUT
	nObjectId : DWORD;
END_VAR
VAR
END_VAR

F_BACnet_GetObjType := TO_INT(SHR((nObjectId AND 16#FFC00000), 22));

END_FUNCTION

// POUs/Local/Objects/FB_BACnet_View
// Structured View Object
{attribute 'enable_dynamic_creation'}
FUNCTION_BLOCK FB_BACnet_View EXTENDS FB_BACnet_Object IMPLEMENTS I_BACnet_View
VAR_INPUT CONSTANT
	{attribute 'parameterCategory':='General'}
	eNodeType : E_BACnet_NodeType := E_BACnet_NodeType.eOrganizational;
END_VAR
VAR
	{region 'Linked Object-List'}
		{attribute 'hide'}
		iFirstChild				: I_BACnet_Object;
		{attribute 'hide'}
		iLastChild				: I_BACnet_Object;
		{attribute 'no_copy'}
		nChildCount				: DINT;
	{endregion}
END_VAR
VAR_STAT
	{region 'Internal'}
		// (BETA) ... Following symbols should be made non-static / thread safe!
		{attribute 'hide'}
		iThisView				: I_BACnet_View;
	{endregion}
END_VAR

SUPER^();

// Unused - Implemented for compatibility reason!
{attribute 'hide'}
METHOD Close
iFirstChild := 0;
iLastChild := 0;
nChildCount := 0;

SUPER^.Close();
END_METHOD

{attribute 'hide'}
METHOD AddObject : BOOL
VAR_INPUT
	iObject			: I_BACnet_Object;
END_VAR
VAR_OUTPUT
	nResultIndex	: DINT;
END_VAR
IF (iObject <> 0) THEN
	iThisView := THIS^;
	
	IF (iObject.Parent = 0) THEN
		fbLogMsg.Show(ADSLOG_MSGTYPE_ERROR, 'AO05', 'No parent defined in child-object!', FALSE);
		
	ELSIF (iObject.Parent <> iThisView) THEN
		fbLogMsg.Show(ADSLOG_MSGTYPE_ERROR, 'AO07', 'Child already assigned to another parent!', FALSE);
		
	ELSE
		IF (FindObject(iObject, nResultIndex)) THEN
			// Child already assigned.
		ELSE
			// Register 'iObject' as a new child in the linked list:
			nResultIndex := nChildCount;
			
			IF (nChildCount = 0) THEN
				iFirstChild := iObject;
			ELSE
				iLastChild.NextSibling := iObject;
				iObject.PrevSibling := iLastChild;
			END_IF
			iLastChild := iObject;
			nChildCount := (nChildCount + 1);
			
			IF (bReady) THEN
				// Register child object:
				View_AddSubordinate(iObject);
			END_IF
		END_IF
		
		AddObject := TRUE;
	END_IF
END_IF
END_METHOD

{attribute 'hide'}
METHOD RemoveObject : BOOL
VAR_INPUT
	iObject			: I_BACnet_Object;
END_VAR
VAR
	_nTemp			: DINT;
	_fbObj			: POINTER TO FB_BACnet_Object;
END_VAR
IF (iObject <> 0) THEN
	iThisView := THIS^;
	
	IF (iObject.Parent = iThisView) AND (FindObject(iObject, _nTemp) <> 0) THEN
		IF (__QUERYPOINTER(iObject, _fbObj)) THEN
			// Remove object from linked object list of current instance:
			_fbObj^.RemoveFromLinkedObjList(iFirstChild, iLastChild);
			nChildCount := (nChildCount-1);
			
			RemoveObject := TRUE;
		END_IF
	END_IF
	
	iObject.Parent := 0;
	iObject.PrevSibling := 0;
	iObject.NextSibling := 0;
END_IF
END_METHOD

METHOD PROTECTED OnObjectStateChanged
VAR
	_iObj			: I_BACnet_Object;
END_VAR
SUPER^.OnObjectStateChanged();

CASE (tState) OF
	TCOM_STATE.TCOM_STATE_PREOP:
		// SyncHandler:
		RequestSyncHandlers(0, 1);
		
	TCOM_STATE.TCOM_STATE_SAFEOP:
		;

	TCOM_STATE.TCOM_STATE_OP:
		SyncProperty(E_BACnetPropIdentifier.PropNodeType, SIZEOF(eNodeType), ADR(eNodeType), 0, eFullSync_InitPLC, FALSE);

		// Add so far registered child objects to subordinate list:
		_iObj := iFirstChild;
		WHILE (_iObj <> 0) DO
			View_AddSubordinate(_iObj);
			_iObj := _iObj.NextSibling;
		END_WHILE

END_CASE
END_METHOD

METHOD FB_init : BOOL
VAR_INPUT
	bInitRetains : BOOL; // if TRUE, the retain variables are initialized (warm start / cold start)
	bInCopyCode : BOOL;  // if TRUE, the instance afterwards gets moved into the copy code (online change)
END_VAR
eObjectType := E_BACnetObjType.ObjStructuredView;
END_METHOD

METHOD FindObject : BOOL
VAR_INPUT
	iObject			: I_BACnet_Object;
END_VAR
VAR_IN_OUT
	nResultIndex	: DINT;
END_VAR
VAR
	_iObj			: I_BACnet_Object;
END_VAR
FindObject := FALSE;

IF (iObject <> 0) THEN
	_iObj := iFirstChild;
	nResultIndex := 0;
	
	WHILE (_iObj <> 0) DO
		IF (_iObj = iObject) THEN
			FindObject := TRUE;
			RETURN;
		ELSE
			nResultIndex := (nResultIndex + 1);
			_iObj := _iObj.NextSibling;
		END_IF
	END_WHILE
END_IF
END_METHOD

END_FUNCTION_BLOCK

// POUs/Helper/[internal]/F_BACnet_AlignedSize
{attribute 'hide'} // [Workaround] Not hidden when lib is included
FUNCTION INTERNAL F_BACnet_AlignedSize : DWORD
VAR_INPUT
	n	: DWORD;
END_VAR
VAR
END_VAR

F_BACnet_AlignedSize := (4*(((n)+3)/4));

END_FUNCTION

// POUs/Helper/[internal]/F_BACnet_SetBitFieldBit
{attribute 'hide'} // [Workaround] Not hidden when lib is included
FUNCTION INTERNAL F_BACnet_SetBitFieldBit : DWORD
VAR_INPUT
	ptrData		:	POINTER TO DWORD;
	bitNbr			:	INT;
END_VAR
VAR
END_VAR

ptrData^ := ptrData^ OR (SHR(DWORD#16#00008000, F_BACnet_BitFieldBit(bitNbr)));
F_BACnet_SetBitFieldBit := ptrData^;

END_FUNCTION

// POUs/Helper/[internal]/F_BACnet_BitFieldBit
{attribute 'hide'} // [Workaround] Not hidden when lib is included
FUNCTION INTERNAL F_BACnet_BitFieldBit : WORD
VAR_INPUT
	bitNbr	:	INT;
END_VAR
VAR
END_VAR

F_BACnet_BitFieldBit := to_word((bitNbr/8) * 8 + (bitNbr MOD 8));

END_FUNCTION

// POUs/Helper/[internal]/String/F_BACnet_EncodeUTF8
{attribute 'hide'} // [Workaround] Not hidden when lib is included
FUNCTION INTERNAL F_BACnet_EncodeUTF8 : UDINT (* actually byte length of the result utf-8 string (maybe longer than cbResult; means overflow) *)
VAR_INPUT
	pString		: POINTER TO BYTE; (* pointer to Win1252 string beginning *)
	nString	: UDINT; (* byte size of string (use SIZEOF - don't use LEN) *)
	pResult		: POINTER TO BYTE; (* pointer to result UTF-8 data area *)
	nResult	: UDINT; (* byte size of result (use SIZEOF - don't use LEN) *)
END_VAR

VAR
	pBy			: POINTER TO BYTE;
	pByArr		: POINTER TO ARRAY[0..3] OF BYTE;
	nCoded		: UINT;
	bOverflow	: BOOL;
END_VAR
(*All VAR_IN_OUT variables have been moved to the end of the declaration due to compatibility reasons*)
VAR_IN_OUT
	nResultLen	: UDINT; (* final resulting string length (<= nResult) *)
END_VAR

pBy			:= pString;
pByArr		:= pResult;
bOverflow	:= FALSE;
F_BACnet_EncodeUTF8 := 0;
nResultLen	:= 0;
(* loop over pString *)
WHILE pBy < (pString + nString) DO
	IF (pBy^ = 0) THEN EXIT; END_IF
	IF bOverflow OR (F_BACnet_EncodeUTF8 + 3 > nResult) THEN
		nCoded := F_BACnet_Win1252ToUtf8(nW1252:=pBy^, pUtf8:=pByArr, bEval:=TRUE);
		IF (NOT bOverflow) AND (F_BACnet_EncodeUTF8 + nCoded <= nResult) THEN
			nCoded := F_BACnet_Win1252ToUtf8(nW1252:=pBy^, pUtf8:=pByArr, bEval:=FALSE);
		ELSE
			bOverflow := TRUE;
		END_IF
	ELSE
		nCoded := F_BACnet_Win1252ToUtf8(nW1252:=pBy^, pUtf8:=pByArr, bEval:=FALSE);
	END_IF
	IF (NOT bOverflow) THEN
		pByArr := pByArr + UINT_TO_UDINT(nCoded);
		nResultLen := F_BACnet_EncodeUTF8 + nCoded;
	END_IF
	F_BACnet_EncodeUTF8 := F_BACnet_EncodeUTF8 + nCoded;
	pBy := pBy + 1;
END_WHILE
(* add zero termination if needed *)
IF (nResultLen < nResult) THEN
	pByArr^[0] := 16#00;
END_IF

END_FUNCTION

// POUs/Helper/[internal]/String/F_BACnet_Win1252ToUtf8
{attribute 'hide'} // [Workaround] Not hidden when lib is included
FUNCTION INTERNAL F_BACnet_Win1252ToUtf8 : UINT(0..3)
VAR_INPUT
	nW1252	: BYTE; (* Win1252 character *)
	pUtf8	: POINTER TO ARRAY[0..2] OF BYTE; (* pointer to target character buffer (utf-8) *)
	bEval	: BOOL; (* TRUE = only evaluate expected coding size (0..3 byte) - but don't write data *)
END_VAR
VAR
	pWord	: POINTER TO ARRAY[0..1] OF BYTE;
	wUCS2	: WORD;
END_VAR
VAR CONSTANT
	cRepl	: BYTE := 16#5F;
END_VAR

(*
	Windows-Codepages
874		Thai
932		Japanisch
936		Vereinfachtes Chinesisch
949		Koreanisch
950		Traditionelles Chinesisch
1250	Mitteleuropäisch
1251	Kyrillisch
1252	Westeuropäisch
1253	Griechisch
1254	Türkisch
1255	Hebräisch
1256	Arabisch
1257	Baltisch
1258	Vietnamesisch
*)
(* check pointer *)
IF (pUtf8 = 0) THEN
	(* null pointer *)
	F_BACnet_Win1252ToUtf8 := 0;
ELSIF (nW1252 <= 16#7F) THEN
	(* basic latin - 1 byte *)
	IF (NOT bEval) THEN
		pUtf8^[0] := nW1252;
	END_IF
	F_BACnet_Win1252ToUtf8 := 1;
ELSE
	(* convert to UCS-2 first *)
	wUCS2 := F_BACnet_Win1252ToUCS2(nW1252:=nW1252, bBE:=FALSE);
	pWord := ADR(wUCS2);
	(* convert used ranges *)
	IF (wUCS2 >= 16#80 AND wUCS2 <= 16#BF) THEN
		(* latin-1 supplement *)
		IF (NOT bEval) THEN
			pUtf8^[0] := 16#C2;
			pUtf8^[1] := pWord^[0];
		END_IF
		F_BACnet_Win1252ToUtf8 := 2;
	ELSIF (wUCS2 >= 16#C0 AND wUCS2 <= 16#FF) THEN
		(* latin-1 supplement *)
		IF (NOT bEval) THEN
			pUtf8^[0] := 16#C3;
			pUtf8^[1] := pWord^[0] - 16#40;
		END_IF
		F_BACnet_Win1252ToUtf8 := 2;
	ELSIF (wUCS2 >= 16#140 AND wUCS2 <= 16#17F) THEN
		(* latin extended A *)
		IF (NOT bEval) THEN
			pUtf8^[0] := 16#C5;
			pUtf8^[1] := pWord^[0] + 16#40;
		END_IF
		F_BACnet_Win1252ToUtf8 := 2;
	ELSIF (wUCS2 >= 16#20A0 AND wUCS2 <= 16#20BF) THEN
		(* currency symbols *)
		IF (NOT bEval) THEN
			pUtf8^[0] := 16#E2;
			pUtf8^[1] := 16#82;
			pUtf8^[2] := pWord^[0];
		END_IF
		F_BACnet_Win1252ToUtf8 := 3;
	ELSE
		(* unsupported *)
		IF (NOT bEval) THEN
			pUtf8^[0] := cRepl;
		END_IF
		F_BACnet_Win1252ToUtf8 := 1;
	END_IF
END_IF

END_FUNCTION

// POUs/Helper/[internal]/String/F_BACnet_Win1252ToUCS2
{attribute 'hide'} // [Workaround] Not hidden when lib is included
FUNCTION INTERNAL F_BACnet_Win1252ToUCS2 : WORD
VAR_INPUT
	nW1252 : BYTE;
	bBE	: BOOL; (* byte-order big endian = TRUE *)
END_VAR
VAR
	pArr : POINTER TO ARRAY[0..1] OF BYTE;
	nBuf : BYTE;
	wUCS2: WORD;
END_VAR

(*
	Windows-Codepages
874		Thai
932		Japanisch
936		Vereinfachtes Chinesisch
949		Koreanisch
950		Traditionelles Chinesisch
1250	Mitteleuropäisch
1251	Kyrillisch
1252	Westeuropäisch
1253	Griechisch
1254	Türkisch
1255	Hebräisch
1256	Arabisch
1257	Baltisch
1258	Vietnamesisch
*)
CASE nW1252 OF
	16#9F: wUCS2 := 16#178;
	16#9C: wUCS2 := 16#153;
	16#8C: wUCS2 := 16#152;
	16#9E: wUCS2 := 16#17E;
	16#8E: wUCS2 := 16#17D;
	16#9A: wUCS2 := 16#161;
	16#8A: wUCS2 := 16#160;
	16#80: wUCS2 := 16#20AC;
	ELSE
	wUCS2 := nW1252;
END_CASE
IF bBE THEN
	pArr := ADR(wUCS2);
	nBuf := pArr^[0];
	pArr^[0] := pArr^[1];
	pArr^[1] := nBuf;
END_IF
F_BACnet_Win1252ToUCS2 := wUCS2;

END_FUNCTION

// POUs/Helper/[internal]/F_BACnet_FilterErrCode
FUNCTION F_BACnet_FilterErrCode : HRESULT
VAR_INPUT
	hResult		: HRESULT;
END_VAR

F_BACnet_FilterErrCode := TO_UINT(hResult) AND 16#FFF;

END_FUNCTION

// POUs/Helper/[internal]/F_BACnet_IsBitFieldBitSet
{attribute 'hide'} // [Workaround] Not hidden when lib is included
FUNCTION INTERNAL F_BACnet_IsBitFieldBitSet : BOOL
VAR_INPUT
	data	:	DWORD;
	bitNbr		:	INT;
END_VAR
VAR
END_VAR

F_BACnet_IsBitFieldBitSet:= (data AND (SHR(DWORD#16#00008000,F_BACnet_BitFieldBit(bitNbr)))) > 0;

END_FUNCTION

// POUs/Helper/[internal]/Scheduler/F_BA_CalendarSchedSize
{attribute 'hide'}
FUNCTION F_BA_CalendarSchedSize : DINT
VAR_IN_OUT
	aCalendar			: ARRAY[*] OF ST_BACnet_SchedCalendar;
END_VAR

F_BA_CalendarSchedSize := (UPPER_BOUND(aCalendar, 1) - LOWER_BOUND(aCalendar, 1) + 1) * SIZEOF(ST_BACnet_SchedCalendar);

END_FUNCTION

// POUs/Helper/[internal]/Scheduler/F_BA_ExceptionSchedSize
{attribute 'hide'}
FUNCTION F_BA_ExceptionSchedSize : DINT
VAR_IN_OUT
	aException			: ARRAY[*] OF ST_BACnet_SchedException;
END_VAR

F_BA_ExceptionSchedSize := (UPPER_BOUND(aException, 1) - LOWER_BOUND(aException, 1) + 1) * SIZEOF(ST_BACnet_SchedException);

END_FUNCTION

// POUs/Helper/[internal]/F_BACnet_EndOf
{attribute 'hide'} // [Workaround] Not hidden when lib is included
FUNCTION INTERNAL F_BACnet_EndOf : POINTER TO BYTE
VAR_INPUT
	 pPtr : POINTER TO BYTE;
	 nSize : DWORD;
END_VAR
VAR
END_VAR

F_BACnet_EndOf:=pPtr+nSize;

END_FUNCTION

// POUs/Helper/[internal]/F_BACnet_NextListElem
{attribute 'hide'} // [Workaround] Not hidden when lib is included
FUNCTION INTERNAL F_BACnet_NextListElem : POINTER TO BYTE
VAR_INPUT
	 pPtr : POINTER TO BYTE;
	 nSize : DWORD;
END_VAR
VAR
END_VAR

IF nSize < 16#80000000 THEN
	F_BACnet_NextListElem:=0;
	RETURN;
END_IF
F_BACnet_NextListElem:=pPtr+F_BACnet_AlignedSize(nSize AND 16#7FFFFFFF)+8;

END_FUNCTION

// POUs/Helper/String/FB_BACnet_StringExtDecode
FUNCTION_BLOCK FB_BACnet_StringExtDecode (* convert UTF-8/UCS2/UCS4/ISO8859-1 to Windows-1252 *)
VAR_INPUT
	pChrStringExt	: POINTER TO ST_BACnet_CharacterStringExt; (* BACnet character string data structure (header and string) *)
	pOutString		: POINTER TO T_MaxString; (* pointer to result buffer (Windows-1252 encoded) *)
	nOutSize		: UDINT; (* byte size *)
END_VAR
VAR_OUTPUT
	bValid			: BOOL; (* Decoding successfull *)
	bOverflow		: BOOL; (* String length overflow (source string too long) *)
	bUnsupported	: BOOL; (* Souce encoding is unsupported (use ReadProp function and decode manually instead) *)
	nLength			: UDINT; (* out character length *)
	eSrcEncoding	: E_BACnet_StringEncodingTypes; (* input encoding *)
END_VAR
VAR
	pText 			: POINTER TO BYTE;
	pByte			: POINTER TO BYTE;
END_VAR

(* preset valid to FALSE *)
bValid := FALSE;
bOverflow := FALSE;
bUnsupported := FALSE;
(* check pointer *)
IF (pChrStringExt = 0) OR (pOutString = 0) THEN
	nLength := 0;
(* check input size *)
ELSIF (nOutSize = 0) THEN
	(* NULL string *)
	bValid := TRUE;
	pOutString^ := '';
	nLength := 0;
	eSrcEncoding := E_BACnet_StringEncodingTypes.eAnsiUtf8;
ELSE
	(* string data available *)
	IF (pChrStringExt^.cookie = 0) THEN
		(* new character string type *)
		nLength			:= UDINT_TO_UINT(pChrStringExt^.strLen);
		eSrcEncoding	:= UDINT_TO_INT(pChrStringExt^.encoding);
		pText			:= ADR(pChrStringExt^.aData);
	ELSE
		(* ASCII/UTF-8 string *)
		nLength			:= F_BACnet_ChrStrExtLen(pChrStringExt^);
		eSrcEncoding	:= E_BACnet_StringEncodingTypes.eAnsiUtf8;
		pText			:= pChrStringExt;
	END_IF

	(* check size *)
	IF (nLength = 0) THEN
		(* no data *)
		bValid := TRUE;
		pOutString^ := '';
	ELSIF (nLength <= nOutSize) THEN
		(* copy to output buffer first *)
		MEMMOVE(destAddr:= pOutString, srcAddr:= pText, n:= nLength);

		(* decode and copy *)
		CASE eSrcEncoding OF

			E_BACnet_StringEncodingTypes.eAnsiUtf8:
				bValid := TRUE;
				nLength := UDINT_TO_UINT(F_BACnet_DecodeUTF8(pOutString, nLength));

			E_BACnet_StringEncodingTypes.eUCS2:
				bValid := TRUE;
				nLength := UDINT_TO_UINT(F_BACnet_DecodeUCS2(pOutString, nLength));

			E_BACnet_StringEncodingTypes.eUCS4:
				bValid := TRUE;
				nLength := UDINT_TO_UINT(F_BACnet_DecodeUCS4(pOutString, nLength));

			E_BACnet_StringEncodingTypes.eISO8859:
				bValid := TRUE;
				(* check if string termination is already part of string *)
				pByte := pOutString + nLength - 1;
				IF (pByte^ = 16#00) THEN
					(* termination already part of string *)
					nLength := nLength - 1;
				ELSE
					(* add string termination *)
					pByte := pOutString + nLength;
					pByte^ := 16#00;
				END_IF

			ELSE
				bUnsupported := TRUE;

		END_CASE
	ELSE
		(* text too long *)
		nLength := 0;
		pOutString^ := '';
		bOverflow := TRUE;
	END_IF
END_IF

END_FUNCTION_BLOCK

// POUs/Helper/[internal]/String/F_BACnet_ChrStrExtLen
{attribute 'hide'} // [Workaround] Not hidden when lib is included
FUNCTION INTERNAL F_BACnet_ChrStrExtLen : UDINT
VAR
	pByte	: POINTER TO BYTE;
	nLen	: UDINT;
END_VAR
(*All VAR_IN_OUT variables have been moved to the end of the declaration due to compatibility reasons*)
VAR_IN_OUT
	stCharStringExt	: ST_BACnet_CharacterStringExt;
END_VAR

pByte := ADR(stCharStringExt);
nLen := SIZEOF(stCharStringExt);
(* check the string type *)
IF (nLen > 4 AND stCharStringExt.cookie = 0) THEN
	(* character string ext. *)
	IF (stCharStringExt.strLen <= SIZEOF(stCharStringExt.aData)) THEN
		(* plausible string length given *)
		F_BACnet_ChrStrExtLen := stCharStringExt.strLen;
		RETURN;
	END_IF
	(* use sizeof, because string length isn't plausible *)
	nLen := SIZEOF(stCharStringExt.aData);
	(* re-adjust pointer *)
	pByte := ADR(stCharStringExt.aData);
END_IF
(* scan zero termination *)
F_BACnet_ChrStrExtLen := 0;
WHILE ((pByte^ <> 0) AND (F_BACnet_ChrStrExtLen < nLen)) DO
	pByte := pByte + 1;
	F_BACnet_ChrStrExtLen := F_BACnet_ChrStrExtLen + 1;
END_WHILE

END_FUNCTION

// POUs/Helper/[internal]/String/F_BACnet_DecodeUTF8
{attribute 'hide'} // [Workaround] Not hidden when lib is included
FUNCTION INTERNAL F_BACnet_DecodeUTF8 : UDINT (* result is the new character length of the string *)
VAR_INPUT
	pString		: POINTER TO BYTE; (* pointer to UTF-8 string beginning *)
	nString	: UDINT; (* byte size of string (use SIZEOF - don't use LEN) *)
END_VAR
VAR
	i			: UDINT;
	pResult		: POINTER TO BYTE;
	pBy			: POINTER TO BYTE;
	pByArr		: POINTER TO ARRAY[0..3] OF BYTE;
END_VAR

pResult	:= pString;
pBy		:= pString;
FOR i := 0 TO nString-1 DO
	pByArr := pBy;
	IF (pByArr^[0] AND 16#F0) = 16#C0 THEN
		IF (pByArr^[1] AND 16#80) = 16#80 THEN
			pResult^ := F_BACnet_Utf8ToWin1252(pByArr, 2);
			pBy := pBy + 2;
		END_IF
	ELSIF (pByArr^[0] AND 16#F0) = 16#E0 THEN
		IF (pByArr^[1] AND 16#80) = 16#80 THEN
			IF (pByArr^[2] AND 16#80) = 16#80 THEN
				pResult^ := F_BACnet_Utf8ToWin1252(pByArr, 3);
				pBy := pBy + 3;
			END_IF
		END_IF
	ELSIF (pByArr^[0] AND 16#F0) = 16#F0 THEN
		IF (pByArr^[1] AND 16#80) = 16#80 THEN
			IF (pByArr^[2] AND 16#80) = 16#80 THEN
				IF (pByArr^[3] AND 16#80) = 16#80 THEN
					pResult^ := F_BACnet_Utf8ToWin1252(pByArr, 4);
					pBy := pBy + 4;
				END_IF
			END_IF
		END_IF
	ELSE
		(* ASCII character *)
		pResult^ := pBy^;
		pBy := pBy + 1;
	END_IF
	(* end-of-string by character *)
	IF (pResult^ = 16#00) THEN
		EXIT;
	END_IF
	(* next character *)
	pResult := pResult + 1;
	(* end-of-string by length *)
	IF (pBy >= (pString + nString)) THEN
		EXIT;
	END_IF
END_FOR
pResult^ := 16#00;
F_BACnet_DecodeUTF8 := pResult - pString;

END_FUNCTION

// POUs/Helper/[internal]/String/F_BACnet_Utf8ToWin1252
{attribute 'hide'} // [Workaround] Not hidden when lib is included
FUNCTION INTERNAL F_BACnet_Utf8ToWin1252 : BYTE
VAR_INPUT
	pUtf8	: POINTER TO BYTE;
	nUtf8	: UDINT; (* byte size of UTF8 character (1...6) *)
END_VAR
VAR
	pArr		: POINTER TO ARRAY[0..5] OF BYTE;
	pWord		: POINTER TO ARRAY[0..1] OF BYTE;
	wUCS2		: WORD;
END_VAR
VAR CONSTANT
	cRepl	: BYTE := 16#5F;
END_VAR

(*
	Windows-Codepages
874		Thai
932		Japanisch
936		Vereinfachtes Chinesisch
949		Koreanisch
950		Traditionelles Chinesisch
1250	Mitteleuropäisch
1251	Kyrillisch
1252	Westeuropäisch
1253	Griechisch
1254	Türkisch
1255	Hebräisch
1256	Arabisch
1257	Baltisch
1258	Vietnamesisch
*)
(* first step - convert to UCS2 *)
pArr := pUtf8;
IF (pArr^[0] <= 16#7F) THEN
	(* basic latin *)
	F_BACnet_Utf8ToWin1252 := pArr^[0];
	RETURN;
ELSIF (nUtf8 >= 2) THEN
	pWord := ADR(wUCS2);
	IF (pArr^[0] = 16#C2) THEN
		(* latin-1 supplement *)
		wUCS2 := pArr^[1];
	ELSIF (pArr^[0] = 16#C3) AND (pArr^[1] <= 16#BF) THEN
		(* latin-1 supplement *)
		wUCS2 := pArr^[1] + 16#40;
	ELSIF (pArr^[0] = 16#C4) AND (pArr^[1] >= 16#80) THEN
		(* latin extended-A *)
		pWord^[1] := 16#01;
		pWord^[0] := pArr^[1] - 16#80;
	ELSIF (pArr^[0] = 16#C5) AND (pArr^[1] >= 16#80) THEN
		(* latin extended-A *)
		pWord^[1] := 16#01;
		pWord^[0] := pArr^[1] - 16#40;
	ELSIF (pArr^[0] = 16#C6) AND (pArr^[1] >= 16#80) THEN
		(* latin extended-B *)
		pWord^[1] := 16#01;
		pWord^[0] := pArr^[1];
	ELSIF (pArr^[0] = 16#C7) AND (pArr^[1] <= 16#BF) THEN
		(* latin extended-B *)
		pWord^[1] := 16#01;
		pWord^[0] := pArr^[1] + 16#40;
	ELSIF (nUtf8 >= 3) THEN
		IF (pArr^[0] = 16#E2) AND (pArr^[1] = 16#82) THEN
			(* currency symbols *)
			pWord^[1] := 16#20;
			pWord^[0] := pArr^[2];
		ELSE
			(* unsupported *)
			F_BACnet_Utf8ToWin1252 := cRepl;
			RETURN;
		END_IF
	ELSE
		(* unsupported *)
		F_BACnet_Utf8ToWin1252 := cRepl;
		RETURN;
	END_IF
	(* convert UCS2 to Windows-1252 *)
	F_BACnet_Utf8ToWin1252 := F_BACnet_UCS2ToWin1252(pWord, FALSE);
	RETURN;
END_IF
(* unsupported *)
F_BACnet_Utf8ToWin1252 := cRepl;

END_FUNCTION

// POUs/Helper/[internal]/String/F_BACnet_UCS2ToWin1252
{attribute 'hide'} // [Workaround] Not hidden when lib is included
FUNCTION INTERNAL F_BACnet_UCS2ToWin1252 : BYTE
VAR_INPUT
	pUCS2 :	POINTER TO WORD;
	bBE	: BOOL; (* byte-order big endian = TRUE *)
END_VAR
VAR
	pArr : POINTER TO ARRAY[0..1] OF BYTE;
	wUCS2: WORD;
END_VAR
VAR CONSTANT
	cRepl	: BYTE := 16#5F;
END_VAR

(*
	Windows-Codepages
874		Thai
932		Japanisch
936		Vereinfachtes Chinesisch
949		Koreanisch
950		Traditionelles Chinesisch
1250	Mitteleuropäisch
1251	Kyrillisch
1252	Westeuropäisch
1253	Griechisch
1254	Türkisch
1255	Hebräisch
1256	Arabisch
1257	Baltisch
1258	Vietnamesisch
*)
pArr := pUCS2;
IF bBE THEN
	wUCS2 := (pArr^[0] * 16#0100) + pArr^[1];
ELSE
	wUCS2 := pUCS2^;
END_IF
CASE wUCS2 OF
	16#178: 	F_BACnet_UCS2ToWin1252 := 16#9F;
	16#153: 	F_BACnet_UCS2ToWin1252 := 16#9C;
	16#152: 	F_BACnet_UCS2ToWin1252 := 16#8C;
	16#17E: 	F_BACnet_UCS2ToWin1252 := 16#9E;
	16#17D: 	F_BACnet_UCS2ToWin1252 := 16#8E;
	16#161: 	F_BACnet_UCS2ToWin1252 := 16#9A;
	16#160: 	F_BACnet_UCS2ToWin1252 := 16#8A;
	16#20AC: 	F_BACnet_UCS2ToWin1252 := 16#80;
	ELSE
		IF wUCS2 <= 16#FF THEN
			F_BACnet_UCS2ToWin1252 := WORD_TO_BYTE(wUCS2);
		ELSE
			F_BACnet_UCS2ToWin1252 := cRepl;
		END_IF
END_CASE

END_FUNCTION

// POUs/Helper/[internal]/String/F_BACnet_DecodeUCS2
{attribute 'hide'} // [Workaround] Not hidden when lib is included
FUNCTION INTERNAL F_BACnet_DecodeUCS2 : UDINT (* result is the new character length of the string *)
VAR_INPUT
	pString		: POINTER TO WORD; (* pointer to UCS2 string beginning *)
	nString	: UDINT; (* byte size of string (use SIZEOF - don't use LEN) *)
END_VAR
VAR
	i		: UDINT;
	pResult	: POINTER TO BYTE;
	pBy		: POINTER TO WORD;
END_VAR

pResult	:= pString;
pBy		:= pString;
FOR i := 0 TO nString-1 DO
	pResult^ := F_BACnet_UCS2ToWin1252(pBy, TRUE);
	pBy := pBy + 2;
	(* end-of-string by character *)
	IF (pResult^ = 16#00) THEN
		EXIT;
	END_IF
	(* next character *)
	pResult := pResult + 1;
	(* end-of-string by length *)
	IF (pBy >= (pString + nString)) THEN
		EXIT;
	END_IF
END_FOR
pResult^ := 16#00;
F_BACnet_DecodeUCS2 := pResult - pString;

END_FUNCTION

// POUs/Helper/[internal]/String/F_BACnet_DecodeUCS4
{attribute 'hide'} // [Workaround] Not hidden when lib is included
FUNCTION INTERNAL F_BACnet_DecodeUCS4 : UDINT (* result is the new character length of the string *)
VAR_INPUT
	pString		: POINTER TO DWORD; (* pointer to UCS4 string beginning *)
	nString	: UDINT; (* byte size of string (use SIZEOF - don't use LEN) *)
END_VAR
VAR
	i		: UDINT;
	pResult	: POINTER TO BYTE;
	pBy		: POINTER TO WORD;
END_VAR

pResult	:= pString;
pBy		:= pString;
FOR i := 0 TO nString-1 DO
	(* byte order big endian *)
	pResult^ := F_BACnet_UCS2ToWin1252(pBy+2, TRUE);
	pBy := pBy + 4;
	(* end-of-string by character *)
	IF (pResult^ = 16#00) THEN
		EXIT;
	END_IF
	(* next character *)
	pResult := pResult + 1;
	(* end-of-string by length *)
	IF (pBy >= (pString + nString)) THEN
		EXIT;
	END_IF
END_FOR
pResult^ := 16#00;
F_BACnet_DecodeUCS4 := pResult - pString;

END_FUNCTION

// POUs/Helper/[internal]/Validation-Functions/F_BACnet_IsObjIdentifierValid
{attribute 'hide'} // [Workaround] Not hidden when lib is included
FUNCTION INTERNAL F_BACnet_IsObjIdentifierValid : BOOL
VAR_INPUT
	tIdentifier		: T_BACnet_ObjectIdentifier;
END_VAR

F_BACnet_IsObjIdentifierValid := ((tIdentifier <> 0) AND_THEN (tIdentifier <> BACnet_Globals.nBACnetObjId_None));

END_FUNCTION

// POUs/Helper/[internal]/Validation-Functions/F_BACnet_IsPriorityValid
{attribute 'hide'} // [Workaround] Not hidden when lib is included
FUNCTION INTERNAL F_BACnet_IsPriorityValid : BOOL
VAR_INPUT
	ePriority		: E_BACnet_Priority;
END_VAR

F_BACnet_IsPriorityValid := ((E_BACnet_Priority.First <= ePriority) AND_THEN (ePriority <= E_BACnet_Priority.Last));

END_FUNCTION

// POUs/Local/Objects/FB_BACnet_AI_Raw
// Analog Input Object
// - Raw communication
{attribute 'pin_presentation_order_outputs' := 'fPresentValue,bEvent,eReliability'}
{attribute 'enable_dynamic_creation'}
FUNCTION_BLOCK FB_BACnet_AI_Raw EXTENDS FB_BACnet_BaseAI
VAR_INPUT
	nRawState					: USINT;			// Raw state
													// - Underrange:	0x01
													// - Overrange:		0x02
													// - Error:			0x04
	nRawValue					: INT;				// Raw value
END_VAR
VAR_INPUT CONSTANT PERSISTENT
	{region 'Variable Parameters'}
		{attribute 'parameterCategory':='Hardware'}
		fResolution : REAL := 0.1;
		{attribute 'parameterCategory':='Hardware'}
		fScaleOffset : REAL := 0
	{endregion};
END_VAR

SUPER^();

METHOD PROTECTED OnObjectStateChanged
CASE (tState) OF
	TCOM_STATE.TCOM_STATE_PREOP:
		// SyncHandler:
		RequestSyncHandlers(1, 4);

	TCOM_STATE.TCOM_STATE_SAFEOP:
		SyncProperty(E_BACnetPropIdentifier.PropPresentValue, SIZEOF(fPresentValue), ADR(fPresentValue), 0, eSync_FromSupplement, TRUE);
		
		SyncProperty(E_BACnetPropIdentifier.PropRawIoStateUSINT, SIZEOF(nRawState), ADR(nRawState), 0, eSync_ToSupplement, TRUE);
		SyncProperty(E_BACnetPropIdentifier.PropRawIoAnalogValueINT, SIZEOF(nRawValue), ADR(nRawValue), 0, eSync_ToSupplement, TRUE);
		
	TCOM_STATE.TCOM_STATE_OP:
		SyncProperty(E_BACnetPropIdentifier.PropResolution, SIZEOF(fResolution), ADR(fResolution), 0, eFullSync_InitPLC, FALSE);
		SyncProperty(E_BACnetPropIdentifier.PropScaleOffset, SIZEOF(fScaleOffset), ADR(fScaleOffset), 0, eFullSync_InitPLC, FALSE);

END_CASE


SUPER^.OnObjectStateChanged();
END_METHOD

END_FUNCTION_BLOCK

// POUs/Local/Objects/[Base]/FB_BACnet_BaseAI
FUNCTION_BLOCK FB_BACnet_BaseAI EXTENDS FB_BACnet_EventObject
VAR_INPUT CONSTANT PERSISTENT
	{region 'Variable Parameters'}
		{attribute 'parameterCategory':='Hardware'}
		{attribute 'TcEncoding':='UTF-8'}
		sDeviceType : STRING;
		{attribute 'parameterCategory':='Hardware'}
		{attribute 'parameterUnit':= '1/100s'}
		nUpdateInterval : UDINT := 5;
		
		{attribute 'parameterCategory':='Value'}
		fMinPresValue : REAL := 0;
		{attribute 'parameterCategory':='Value'}
		fMaxPresValue : REAL := 100;
		{attribute 'parameterCategory':='Value'}
		fFaultDeadband : REAL := 0.0;
		{attribute 'parameterCategory':='Value'}
		bOutOfService : BOOL;
		{attribute 'parameterCategory':='Value'}
		fCOVIncrement : REAL := 0.1;
		{attribute 'parameterCategory':='Value'}
		nAvgFilterCycles : UDINT := 0;
		{attribute 'parameterCategory':='Value'}
		eUnit : E_BA_Unit := E_BA_Unit.eOther_NoUnits;
		
		{attribute 'parameterCategory':='EventConfig'}
		bLowLimitEnable : BOOL := FALSE;
		{attribute 'parameterCategory':='EventConfig'}
		fLowLimitValue : REAL;
		{attribute 'parameterCategory':='EventConfig'}
		bHighLimitEnable : BOOL := FALSE;
		{attribute 'parameterCategory':='EventConfig'}
		fHighLimitValue : REAL;
		{attribute 'parameterCategory':='EventConfig'}
		fDeadband : REAL := 0.0;
	{endregion}
END_VAR
VAR_OUTPUT
	fPresentValue	: REAL;
END_VAR

SUPER^();

METHOD PROTECTED OnObjectStateChanged
SUPER^.OnObjectStateChanged();

CASE (tState) OF
	TCOM_STATE.TCOM_STATE_PREOP:
		// SyncHandler:
		RequestSyncHandlers(0, 14);
		
		// Ensure UTF-8 Encoding:
		F_BA_EnsureUTF8(ADR(sDeviceType), SIZEOF(sDeviceType));
		
	TCOM_STATE.TCOM_STATE_SAFEOP:
		;
		
	TCOM_STATE.TCOM_STATE_OP:
		SyncProperty(E_BACnetPropIdentifier.PropDeviceType, SIZEOF(sDeviceType), ADR(sDeviceType), 0, eFullSync_InitPLC, FALSE);
		SyncProperty(E_BACnetPropIdentifier.PropUpdateInterval, SIZEOF(nUpdateInterval), ADR(nUpdateInterval), 0, eFullSync_InitPLC, FALSE);
		SyncProperty(E_BACnetPropIdentifier.PropUnits, SIZEOF(eUnit), ADR(eUnit), 0, eFullSync_InitPLC, FALSE);
		SyncProperty(E_BACnetPropIdentifier.PropMinPresValue, SIZEOF(fMinPresValue), ADR(fMinPresValue), 0, eFullSync_InitPLC, FALSE);
		SyncProperty(E_BACnetPropIdentifier.PropMaxPresValue, SIZEOF(fMaxPresValue), ADR(fMaxPresValue), 0, eFullSync_InitPLC, FALSE);
		SyncProperty(E_BACnetPropIdentifier.PropFaultDeadband, SIZEOF(fFaultDeadband), ADR(fFaultDeadband), 0, eFullSync_InitPLC, FALSE);
		SyncProperty(E_BACnetPropIdentifier.PropOutOfService, SIZEOF(bOutOfService), ADR(bOutOfService), 0, eFullSync_InitPLC, FALSE);
		SyncProperty(E_BACnetPropIdentifier.PropCovIncrement, SIZEOF(fCOVIncrement), ADR(fCOVIncrement), 0, eFullSync_InitPLC, FALSE);
		SyncProperty(E_BACnetPropIdentifier.PropAvgFilterCycles, SIZEOF(nAvgFilterCycles), ADR(nAvgFilterCycles), 0, eFullSync_InitPLC, FALSE);
		SyncPropertyIdx(E_BACnetPropIdentifier.PropLimitEnable, SIZEOF(BOOL), ADR(bHighLimitEnable), E_BACnet_LimitEnableBits.eHighLimit, 0, eFullSync_InitPLC, FALSE);	
		SyncPropertyIdx(E_BACnetPropIdentifier.PropLimitEnable, SIZEOF(BOOL), ADR(bLowLimitEnable), E_BACnet_LimitEnableBits.eLowLimit, 0, eFullSync_InitPLC, FALSE);
		SyncProperty(E_BACnetPropIdentifier.PropHighLimit, SIZEOF(fHighLimitValue), ADR(fHighLimitValue), 0, eFullSync_InitPLC, FALSE);
		SyncProperty(E_BACnetPropIdentifier.PropLowLimit, SIZEOF(fLowLimitValue), ADR(fLowLimitValue), 0, eFullSync_InitPLC, FALSE);
		SyncProperty(E_BACnetPropIdentifier.PropDeadband, SIZEOF(fDeadband), ADR(fDeadband), 0, eFullSync_InitPLC, FALSE);
		
END_CASE
END_METHOD

METHOD FB_init : BOOL
VAR_INPUT
	bInitRetains : BOOL; // if TRUE, the retain variables are initialized (warm start / cold start)
	bInCopyCode : BOOL;  // if TRUE, the instance afterwards gets moved into the copy code (online change)
END_VAR
eObjectType := E_BACnetObjType.ObjAnalogInput;
END_METHOD

END_FUNCTION_BLOCK

// POUs/Local/Objects/[Base]/Basic/FB_BACnet_EventObject
FUNCTION_BLOCK FB_BACnet_EventObject EXTENDS FB_BACnet_Object
VAR_INPUT CONSTANT PERSISTENT
	{region 'Variable Parameters'}
		{attribute 'parameterCategory':='EventConfig'}
		bEventDetectionEnable : BOOL := TRUE;
		
		{attribute 'parameterCategory':='EventConfig'}
		nNotificationClass : UDINT;
		{attribute 'parameterCategory':='EventConfig'}
		eNotifyType : E_BACnet_NotifyType := E_BACnet_NotifyType.eAlarm;
		{attribute 'parameterCategory':='EventConfig'}
		aEventEnable : T_BACnet_EventTransitions;
		{attribute 'parameterCategory':='EventConfig'}
		aEventMessageTextsConfig : T_BACnet_EventTransitionTexts;
		{attribute 'parameterCategory':='EventConfig'}
		nTimeDelay : UDINT;
		{attribute 'parameterCategory':='EventConfig'}
		nTimeDelayNormal : UDINT;
	{endregion}
END_VAR
VAR_INPUT CONSTANT
	{region 'Operational Parameters'}
		{attribute 'parameterCategory':='Event'}
		bAcknowledgeRm : BOOL;														// Acknowledge outstanding event transition states (from remote via parameter).
	{endregion}
END_VAR
VAR_OUTPUT
	bEvent						: BOOL;												// Indicates an active event
	eReliability				: E_BA_Reliability;
END_VAR
VAR
	{region 'Event'}
		stStatusFlags			: ST_BA_StatusFlags;
		stAckedTransitions		: ST_BA_EventTransitions;

		eEventState				: E_BACnet_EventState;
	{endregion}
	{region 'Misc'}
		rAckPLCTrig				: R_TRIG;
	{endregion}
	{region 'Internal'}
		{attribute 'hide'}
		_bEnEvtDetect			: BOOL;
	{endregion}
END_VAR

rAckPLCTrig();
IF (rAckPLCTrig.Q) THEN
	// Acknowledge all event states:
	Acknowledge(E_BA_EventTransition.Invalid, BACnet_Param.sEvtMgmt_AckMsgPLC);
END_IF
IF bAcknowledgeRm THEN
	bAcknowledgeRm := FALSE;
	// Acknowledge all event states:
	Acknowledge(E_BA_EventTransition.Invalid, BACnet_Param.sEvtMgmt_AckMsgRemote);
END_IF

SUPER^();

bEvent := F_BA_IsDisturbed(stStatusFlags);

METHOD PROTECTED OnObjectStateChanged
SUPER^.OnObjectStateChanged();

CASE (tState) OF
	TCOM_STATE.TCOM_STATE_PREOP:
		// SyncHandler:
		RequestSyncHandlers(9, 11);
		
		// Properties:
		EnableProperty(E_BACnetPropIdentifier.PropEventAlgorithmInhibit, FALSE);
		EnableProperty(E_BACnetPropIdentifier.PropReliabilityEvaluationInhibit, FALSE);
		EnableProperty(E_BACnetPropIdentifier.PropEventDetectionEnable, TRUE);
		
		// Ensure UTF-8 Encoding:
		F_BA_EnsureUTF8Array(ADR(aEventMessageTextsConfig), SIZEOF(aEventMessageTextsConfig[1]), TO_DINT(E_BA_EventTransition.Count));
		
	TCOM_STATE.TCOM_STATE_SAFEOP:
		;
	
	TCOM_STATE.TCOM_STATE_OP:
		ConcatTitle(aEventMessageTextsConfig[E_BA_EventTransition.eToOffnormal], sDescription, BACnet_Param.sSeparator_EventMessageText);
		ConcatTitle(aEventMessageTextsConfig[E_BA_EventTransition.eToFault], sDescription, BACnet_Param.sSeparator_EventMessageText);
		ConcatTitle(aEventMessageTextsConfig[E_BA_EventTransition.eToNormal], sDescription, BACnet_Param.sSeparator_EventMessageText);
		
		// Disable EventDetection at initialization to prevent unacknowledged event states:
		_bEnEvtDetect := bEventDetectionEnable;
		bEventDetectionEnable := FALSE;
		
		// Synchronize:
		SyncProperty(E_BACnetPropIdentifier.PropEventDetectionEnable, SIZEOF(bEventDetectionEnable), ADR(bEventDetectionEnable), 0, eFullSync_InitPLC, FALSE);
		SyncProperty(E_BACnetPropIdentifier.PropNotificationClass, SIZEOF(nNotificationClass), ADR(nNotificationClass), 0, eFullSync_InitPLC, FALSE);
		SyncProperty(E_BACnetPropIdentifier.PropNotifyType, SIZEOF(eNotifyType), ADR(eNotifyType), 0, eFullSync_InitPLC, FALSE);
		SyncPropertyIdx(E_BACnetPropIdentifier.PropEventEnable, SIZEOF(BOOL), ADR(aEventEnable[E_BA_EventTransition.eToOffnormal]), E_BACnet_EventTransitionBits.eToOffnormal, 0, eFullSync_InitPLC, FALSE);	
		SyncPropertyIdx(E_BACnetPropIdentifier.PropEventEnable, SIZEOF(BOOL), ADR(aEventEnable[E_BA_EventTransition.eToFault]), E_BACnet_EventTransitionBits.eToFault, 0, eFullSync_InitPLC, FALSE);	
		SyncPropertyIdx(E_BACnetPropIdentifier.PropEventEnable, SIZEOF(BOOL), ADR(aEventEnable[E_BA_EventTransition.eToNormal]), E_BACnet_EventTransitionBits.eToNormal, 0, eFullSync_InitPLC, FALSE);
		SyncPropertyIdx(E_BACnetPropIdentifier.PropEventMessageTextsConfig, SIZEOF(T_MaxString), ADR(aEventMessageTextsConfig[E_BA_EventTransition.eToOffnormal]), (E_BACnet_EventTransitionBits.eToOffnormal+1), 0, eFullSync_InitPLC, FALSE);
		SyncPropertyIdx(E_BACnetPropIdentifier.PropEventMessageTextsConfig, SIZEOF(T_MaxString), ADR(aEventMessageTextsConfig[E_BA_EventTransition.eToFault]), (E_BACnet_EventTransitionBits.eToFault+1), 0, eFullSync_InitPLC, FALSE);
		SyncPropertyIdx(E_BACnetPropIdentifier.PropEventMessageTextsConfig, SIZEOF(T_MaxString), ADR(aEventMessageTextsConfig[E_BA_EventTransition.eToNormal]), (E_BACnet_EventTransitionBits.eToNormal+1), 0, eFullSync_InitPLC, FALSE);
		
		IF (eObjectType <> E_BACnetObjType.ObjTrendLog) AND (eObjectType <> E_BACnetObjType.ObjTrendLogMultiple) THEN
			IF (eObjectType <> E_BACnetObjType.ObjEventEnrollment) THEN
				SyncProperty(E_BACnetPropIdentifier.PropTimeDelay, SIZEOF(nTimeDelay), ADR(nTimeDelay), 0, eFullSync_InitPLC, FALSE);
			END_IF
			SyncProperty(E_BACnetPropIdentifier.PropTimeDelayNormal, SIZEOF(nTimeDelayNormal), ADR(nTimeDelayNormal), 0, eFullSync_InitPLC, FALSE);
		END_IF
		
		SyncPropertyIdx(E_BACnetPropIdentifier.PropStatusFlags, SIZEOF(BOOL), ADR(stStatusFlags.bOverridden), E_BACnet_StatusFlags.eOverridden, 0, eSync_FromSupplement, FALSE);	
		SyncPropertyIdx(E_BACnetPropIdentifier.PropStatusFlags, SIZEOF(BOOL), ADR(stStatusFlags.bOutOfService), E_BACnet_StatusFlags.eOutOfService, 0, eSync_FromSupplement, FALSE);	
		SyncPropertyIdx(E_BACnetPropIdentifier.PropStatusFlags, SIZEOF(BOOL), ADR(stStatusFlags.bFault), E_BACnet_StatusFlags.eFault, 0, eSync_FromSupplement, FALSE);	
		SyncPropertyIdx(E_BACnetPropIdentifier.PropStatusFlags, SIZEOF(BOOL), ADR(stStatusFlags.bInAlarm), E_BACnet_StatusFlags.eInAlarm, 0, eSync_FromSupplement, FALSE);
		SyncPropertyIdx(E_BACnetPropIdentifier.PropAckedTransitions, SIZEOF(BOOL), ADR(stAckedTransitions.bToOffnormal), E_BACnet_EventTransitionBits.eToOffnormal, 0, eSync_FromSupplement, FALSE);	
		SyncPropertyIdx(E_BACnetPropIdentifier.PropAckedTransitions, SIZEOF(BOOL), ADR(stAckedTransitions.bToFault), E_BACnet_EventTransitionBits.eToFault, 0, eSync_FromSupplement, FALSE);	
		SyncPropertyIdx(E_BACnetPropIdentifier.PropAckedTransitions, SIZEOF(BOOL), ADR(stAckedTransitions.bToNormal), E_BACnet_EventTransitionBits.eToNormal, 0, eSync_FromSupplement, FALSE);	
		SyncProperty(E_BACnetPropIdentifier.PropReliability, SIZEOF(eReliability), ADR(eReliability), 0, eSync_FromSupplement, FALSE);
		SyncProperty(E_BACnetPropIdentifier.PropEventState, SIZEOF(eEventState), ADR(eEventState), 0,  eSync_FromSupplement, FALSE);
		
END_CASE
END_METHOD

// Called on first operational cycle after initialization.
METHOD PROTECTED OnPostInit
// Restore previous mode:
bEventDetectionEnable := _bEnEvtDetect;

SUPER^.OnPostInit();
END_METHOD

METHOD FB_init : BOOL
VAR_INPUT
	bInitRetains : BOOL; // if TRUE, the retain variables are initialized (warm start / cold start)
	bInCopyCode : BOOL;  // if TRUE, the instance afterwards gets moved into the copy code (online change)
END_VAR
IF (bInitRetains) THEN
	// Indicate inheritance of event message texts as default:
	aEventMessageTextsConfig[E_BA_EventTransition.eToOffnormal] := CONCAT(BACnet_Globals.sCmd_ConcatTitle, 'To Off-Normal');
	aEventMessageTextsConfig[E_BA_EventTransition.eToFault] := CONCAT(BACnet_Globals.sCmd_ConcatTitle, 'To Fault');
	aEventMessageTextsConfig[E_BA_EventTransition.eToNormal] := CONCAT(BACnet_Globals.sCmd_ConcatTitle, 'To Normal');
END_IF
END_METHOD

// Acknowledge via Property.
// > This property is triggered (Only rising edges acknowledges current instance!)
PROPERTY AcknowledgePLC : BOOL
GET
AcknowledgePLC := rAckPLCTrig.CLK;
END_GET
SET
rAckPLCTrig.CLK := AcknowledgePLC;
END_SET
END_PROPERTY

PROPERTY AcknowledgeRm : BOOL
GET
AcknowledgeRm := bAcknowledgeRm;
END_GET
SET
bAcknowledgeRm := AcknowledgeRm;
END_SET
END_PROPERTY

PROPERTY IsReliable : BOOL
GET
IsReliable := (eReliability = E_BA_Reliability.eNoFaultDetected) AND (NOT stStatusFlags.bOverridden) AND (NOT stStatusFlags.bOutOfService);
END_GET
END_PROPERTY

PROPERTY AckedTransitions : ST_BA_EventTransitions
GET
AckedTransitions := stAckedTransitions;
END_GET
END_PROPERTY

PROPERTY EventState : E_BACnet_EventState
GET
EventState := eEventState;
END_GET
END_PROPERTY

PROPERTY StatusFlags : ST_BA_StatusFlags
GET
StatusFlags := stStatusFlags;
END_GET
END_PROPERTY

END_FUNCTION_BLOCK

// POUs/Local/Objects/FB_BACnet_AO_Raw
// Analog Output Object
// - Raw communication
// - 1 Priority
{attribute 'pin_presentation_order_outputs' := 'fPresentValue,bEvent,eReliability'}
{attribute 'enable_dynamic_creation'}
FUNCTION_BLOCK FB_BACnet_AO_Raw EXTENDS FB_BACnet_BaseAO
VAR_INPUT
	bRawOverridden				: BOOL;				// Raw overridden
END_VAR
VAR_OUTPUT
	nRawValue					: INT;				// Raw value
END_VAR

IF (bReady) THEN
	// Overridden IO:
	_bOverriddenValue := bRawOverridden;
END_IF

SUPER^();

METHOD PROTECTED OnObjectStateChanged
SUPER^.OnObjectStateChanged();

CASE (tState) OF
	TCOM_STATE.TCOM_STATE_PREOP:
		// SyncHandler:
		RequestSyncHandlers(1, 0);

	TCOM_STATE.TCOM_STATE_SAFEOP:
		SyncProperty(E_BACnetPropIdentifier.PropRawIoAnalogValueINT, SIZEOF(nRawValue), ADR(nRawValue), 0, eSync_FromSupplement, TRUE);
		
	TCOM_STATE.TCOM_STATE_OP:
		;

END_CASE
END_METHOD

END_FUNCTION_BLOCK

// POUs/Local/Objects/[Base]/FB_BACnet_BaseAO
FUNCTION_BLOCK FB_BACnet_BaseAO EXTENDS FB_BACnet_EventObject
VAR_INPUT
	bEnPgm					: BOOL;
	fValPgm					: REAL;
END_VAR
VAR_INPUT CONSTANT PERSISTENT
	{region 'Variable Parameters'}
		{attribute 'parameterCategory':='Hardware'}
		{attribute 'TcEncoding':='UTF-8'}
		sDeviceType : STRING;
		{attribute 'parameterCategory':='Hardware'}
		fResolution : REAL := 0.1;
		{attribute 'parameterCategory':='Hardware'}
		fScaleOffset : REAL := 0;
		
		{attribute 'parameterCategory':='Value'}
		fMinPresValue : REAL := 0;
		{attribute 'parameterCategory':='Value'}
		fMaxPresValue : REAL := 100;
		{attribute 'parameterCategory':='Value'}
		fRelinquishDefault : REAL;
		{attribute 'parameterCategory':='Value'}
		bOutOfService : BOOL;
		{attribute 'parameterCategory':='Value'}
		fCOVIncrement : REAL := 0.1;
		{attribute 'parameterCategory':='Value'}
		eUnit : E_BA_Unit := E_BA_Unit.eOther_NoUnits;
		
		{attribute 'parameterCategory':='EventConfig'}
		bLowLimitEnable : BOOL := FALSE;
		{attribute 'parameterCategory':='EventConfig'}
		fLowLimitValue : REAL;
		{attribute 'parameterCategory':='EventConfig'}
		bHighLimitEnable : BOOL := FALSE;
		{attribute 'parameterCategory':='EventConfig'}
		fHighLimitValue : REAL;
		{attribute 'parameterCategory':='EventConfig'}
		fDeadband : REAL := 0.0;
	{endregion}
END_VAR
VAR_OUTPUT
	fPresentValue			: REAL;
	eActivePrio				: E_BACnet_Priority;			// Indicates the currently active priority of the priority array
END_VAR
VAR
	{region 'Internal'}
		_bOverriddenValue	: BOOL;
	{endregion}
END_VAR

SUPER^();

METHOD PROTECTED OnObjectStateChanged
SUPER^.OnObjectStateChanged();

CASE (tState) OF
	TCOM_STATE.TCOM_STATE_PREOP:
		// SyncHandler:
		RequestSyncHandlers(1, 16);
		
		// Ensure UTF-8 Encoding:
		F_BA_EnsureUTF8(ADR(sDeviceType), SIZEOF(sDeviceType));
		
	TCOM_STATE.TCOM_STATE_SAFEOP:
		SyncPropertyPvPrio(E_BACnetPropIdentifier.PropPresentValue, SIZEOF(fValPgm), ADR(fValPgm), ADR(bEnPgm), BACnet_Param.ePrio_Program, 0, eFullSync_InitPLC, TRUE);
		
		SyncProperty(E_BACnetPropIdentifier.PropPresentValue, SIZEOF(fPresentValue), ADR(fPresentValue), 0, eSync_FromSupplement, TRUE);
		SyncProperty(E_BACnetPropIdentifier.PropCurrentlyActivePriority, SIZEOF(eActivePrio), ADR(eActivePrio), 0, eSync_FromSupplement, TRUE);
		
	TCOM_STATE.TCOM_STATE_OP:
		SyncProperty(E_BACnetPropIdentifier.PropResolution, SIZEOF(fResolution), ADR(fResolution), 0, eFullSync_InitPLC, FALSE);
		SyncProperty(E_BACnetPropIdentifier.PropScaleOffset, SIZEOF(fScaleOffset), ADR(fScaleOffset), 0, eFullSync_InitPLC, FALSE);
		SyncProperty(E_BACnetPropIdentifier.PropDeviceType, SIZEOF(sDeviceType), ADR(sDeviceType), 0, eFullSync_InitPLC, FALSE);
		SyncProperty(E_BACnetPropIdentifier.PropUnits, SIZEOF(eUnit), ADR(eUnit), 0, eFullSync_InitPLC, FALSE);
		SyncProperty(E_BACnetPropIdentifier.PropMinPresValue, SIZEOF(fMinPresValue), ADR(fMinPresValue), 0, eFullSync_InitPLC, FALSE);
		SyncProperty(E_BACnetPropIdentifier.PropMaxPresValue, SIZEOF(fMaxPresValue), ADR(fMaxPresValue), 0, eFullSync_InitPLC, FALSE);
		SyncPropertyIdx(E_BACnetPropIdentifier.PropLimitEnable, SIZEOF(BOOL), ADR(bHighLimitEnable), E_BACnet_LimitEnableBits.eHighLimit, 0, eFullSync_InitPLC, FALSE);	
		SyncPropertyIdx(E_BACnetPropIdentifier.PropLimitEnable, SIZEOF(BOOL), ADR(bLowLimitEnable), E_BACnet_LimitEnableBits.eLowLimit, 0, eFullSync_InitPLC, FALSE);
		SyncProperty(E_BACnetPropIdentifier.PropHighLimit, SIZEOF(fHighLimitValue), ADR(fHighLimitValue), 0, eFullSync_InitPLC, FALSE);
		SyncProperty(E_BACnetPropIdentifier.PropLowLimit, SIZEOF(fLowLimitValue), ADR(fLowLimitValue), 0, eFullSync_InitPLC, FALSE);
		SyncProperty(E_BACnetPropIdentifier.PropDeadband, SIZEOF(fDeadband), ADR(fDeadband), 0, eFullSync_InitPLC, FALSE);
		SyncProperty(E_BACnetPropIdentifier.PropRelinquishDefault, SIZEOF(fRelinquishDefault), ADR(fRelinquishDefault), 0, eFullSync_InitPLC, FALSE);
		SyncProperty(E_BACnetPropIdentifier.PropOutOfService, SIZEOF(bOutOfService), ADR(bOutOfService), 0, eFullSync_InitPLC, FALSE);
		SyncProperty(E_BACnetPropIdentifier.PropCovIncrement, SIZEOF(fCOVIncrement), ADR(fCOVIncrement), 0, eFullSync_InitPLC, FALSE);
		
		SyncProperty(E_BACnetPropIdentifier.PropRawIoStateOverride, SIZEOF(_bOverriddenValue), ADR(_bOverriddenValue), 0, eSync_ToSupplement, FALSE);
		
END_CASE
END_METHOD

METHOD FB_init : BOOL
VAR_INPUT
	bInitRetains : BOOL; // if TRUE, the retain variables are initialized (warm start / cold start)
	bInCopyCode : BOOL;  // if TRUE, the instance afterwards gets moved into the copy code (online change)
END_VAR
eObjectType := E_BACnetObjType.ObjAnalogOutput;
END_METHOD

PROPERTY ActivePrio : E_BACnet_Priority
GET
ActivePrio := eActivePrio;
END_GET
END_PROPERTY

END_FUNCTION_BLOCK

// POUs/Local/Objects/5P/FB_BACnet_AO_Raw5P
// Analog Output Object
// - Raw communication
// - 5 Priorities
{attribute 'pin_presentation_order_inputs' := 'bEnSfty,fValSfty,bEnCrit,fValCrit,bEnManLoc,fValManLoc,bEnPgm,fValPgm'}
{attribute 'pin_presentation_order_outputs' := 'fPresentValue,eActivePrio,bEvent,eReliability'}
{attribute 'enable_dynamic_creation'}
FUNCTION_BLOCK FB_BACnet_AO_Raw5P EXTENDS FB_BACnet_AO_Raw
VAR_INPUT
	bEnSfty					: BOOL;
	fValSfty				: REAL;
	bEnCrit					: BOOL;
	fValCrit				: REAL;
	bEnManLoc				: BOOL;
	fValManLoc				: REAL;
END_VAR
VAR_INPUT CONSTANT PERSISTENT
	{region 'Operational Parameters'}
		{attribute 'parameterCategory':='Manual'}
		bEnManualRm : BOOL;
		{attribute 'parameterCategory':='Manual'}
		fValManualRm : REAL;
	{endregion}
END_VAR

SUPER^();

METHOD PROTECTED OnObjectStateChanged
SUPER^.OnObjectStateChanged();

CASE (tState) OF
	TCOM_STATE.TCOM_STATE_PREOP:
		// SyncHandler:
		RequestSyncHandlers(1, 4);
		
	TCOM_STATE.TCOM_STATE_SAFEOP:
		SyncPropertyPvPrio(E_BACnetPropIdentifier.PropPresentValue, SIZEOF(fValSfty), ADR(fValSfty), ADR(bEnSfty), BACnet_Param.ePrio_LifeSafety, 0, eFullSync_InitPLC, TRUE);
		SyncPropertyPvPrio(E_BACnetPropIdentifier.PropPresentValue, SIZEOF(fValCrit), ADR(fValCrit), ADR(bEnCrit), BACnet_Param.ePrio_Critical, 0, eFullSync_InitPLC, TRUE);
		SyncPropertyPvPrio(E_BACnetPropIdentifier.PropPresentValue, SIZEOF(fValManLoc), ADR(fValManLoc), ADR(bEnManLoc), BACnet_Param.ePrio_ManLocal, 0, eFullSync_InitPLC, TRUE);
		SyncPropertyPvPrio(E_BACnetPropIdentifier.PropPresentValue, SIZEOF(fValManualRm), ADR(fValManualRm), ADR(bEnManualRm), BACnet_Param.ePrio_ManRemote, 0, eFullSync_InitPLC, TRUE);
		
	TCOM_STATE.TCOM_STATE_OP:
		;
		
END_CASE
END_METHOD

PROPERTY EnManualRm : BOOL
GET
EnManualRm := bEnManualRm;
END_GET
SET
bEnManualRm := EnManualRm;
END_SET
END_PROPERTY

PROPERTY ValManualRm : REAL
GET
ValManualRm := fValManualRm;
END_GET
SET
fValManualRm := ValManualRm;
END_SET
END_PROPERTY

END_FUNCTION_BLOCK

// POUs/Local/Objects/FB_BACnet_AV
// Analog Value Object
// - 1 Priority
{attribute 'enable_dynamic_creation'}
FUNCTION_BLOCK FB_BACnet_AV EXTENDS FB_BACnet_EventObject
VAR_INPUT
	bEnPgm			: BOOL;
	fValPgm			: REAL;
END_VAR
VAR_INPUT CONSTANT PERSISTENT
	{region 'Variable Parameters'}
		{attribute 'parameterCategory':='Value'}
		fRelinquishDefault : REAL;
		{attribute 'parameterCategory':='Value'}
		bOutOfService : BOOL;
		{attribute 'parameterCategory':='Value'}
		fCOVIncrement : REAL := 0.1;
		{attribute 'parameterCategory':='Value'}
		eUnit : E_BA_Unit := E_BA_Unit.eOther_NoUnits;
		
		{attribute 'parameterCategory':='EventConfig'}
		bLowLimitEnable : BOOL := FALSE;
		{attribute 'parameterCategory':='EventConfig'}
		fLowLimitValue : REAL;
		{attribute 'parameterCategory':='EventConfig'}
		bHighLimitEnable : BOOL := FALSE;
		{attribute 'parameterCategory':='EventConfig'}
		fHighLimitValue : REAL;
		{attribute 'parameterCategory':='EventConfig'}
		fDeadband : REAL := 0.0;
	{endregion}
END_VAR
VAR_OUTPUT
	fPresentValue	: REAL;
	eActivePrio		: E_BACnet_Priority;			// Indicates the currently active priority of the priority array
END_VAR

SUPER^();

METHOD PROTECTED OnObjectStateChanged
SUPER^.OnObjectStateChanged();

CASE (tState) OF
	TCOM_STATE.TCOM_STATE_PREOP:
		// SyncHandler:
		RequestSyncHandlers(1, 9);
		
		// DisableProperty(E_BACnetPropIdentifier.PropDeviceType);

	TCOM_STATE.TCOM_STATE_SAFEOP:
		SyncPropertyPvPrio(E_BACnetPropIdentifier.PropPresentValue, SIZEOF(fValPgm), ADR(fValPgm), ADR(bEnPgm), BACnet_Param.ePrio_Program, 0, eFullSync_InitPLC, TRUE);
		
		SyncProperty(E_BACnetPropIdentifier.PropPresentValue, SIZEOF(fPresentValue), ADR(fPresentValue), 0, eSync_FromSupplement, TRUE);
		SyncProperty(E_BACnetPropIdentifier.PropCurrentlyActivePriority, SIZEOF(eActivePrio), ADR(eActivePrio), 0, eSync_FromSupplement, TRUE);
		
	TCOM_STATE.TCOM_STATE_OP:
		SyncProperty(E_BACnetPropIdentifier.PropUnits, SIZEOF(eUnit), ADR(eUnit), 0, eFullSync_InitPLC, FALSE);
		SyncPropertyIdx(E_BACnetPropIdentifier.PropLimitEnable, SIZEOF(BOOL), ADR(bHighLimitEnable), E_BACnet_LimitEnableBits.eHighLimit, 0, eFullSync_InitPLC, FALSE);	
		SyncPropertyIdx(E_BACnetPropIdentifier.PropLimitEnable, SIZEOF(BOOL), ADR(bLowLimitEnable), E_BACnet_LimitEnableBits.eLowLimit, 0, eFullSync_InitPLC, FALSE);
		SyncProperty(E_BACnetPropIdentifier.PropHighLimit, SIZEOF(fHighLimitValue), ADR(fHighLimitValue), 0, eFullSync_InitPLC, FALSE);
		SyncProperty(E_BACnetPropIdentifier.PropLowLimit, SIZEOF(fLowLimitValue), ADR(fLowLimitValue), 0, eFullSync_InitPLC, FALSE);
		SyncProperty(E_BACnetPropIdentifier.PropDeadband, SIZEOF(fDeadband), ADR(fDeadband), 0, eFullSync_InitPLC, FALSE);
		SyncProperty(E_BACnetPropIdentifier.PropRelinquishDefault, SIZEOF(fRelinquishDefault), ADR(fRelinquishDefault), 0, eFullSync_InitPLC, FALSE);
		SyncProperty(E_BACnetPropIdentifier.PropOutOfService, SIZEOF(bOutOfService), ADR(bOutOfService), 0, eFullSync_InitPLC, FALSE);
		SyncProperty(E_BACnetPropIdentifier.PropCovIncrement, SIZEOF(fCOVIncrement), ADR(fCOVIncrement), 0, eFullSync_InitPLC, FALSE);
		
END_CASE
END_METHOD

METHOD FB_init : BOOL
VAR_INPUT
	bInitRetains : BOOL; // if TRUE, the retain variables are initialized (warm start / cold start)
	bInCopyCode : BOOL;  // if TRUE, the instance afterwards gets moved into the copy code (online change)
END_VAR
eObjectType := E_BACnetObjType.ObjAnalogValue;
END_METHOD

PROPERTY ActivePrio : E_BACnet_Priority
GET
ActivePrio := eActivePrio;
END_GET
END_PROPERTY

END_FUNCTION_BLOCK

// POUs/Local/Objects/5P/FB_BACnet_AV_5P
// Analog Value Object
// - 5 Priorities
{attribute 'pin_presentation_order_inputs' := 'bEnSfty,fValSfty,bEnCrit,fValCrit,bEnManLoc,fValManLoc,bEnPgm,fValPgm'}
{attribute 'pin_presentation_order_outputs' := 'fPresentValue,eActivePrio,bEvent,eReliability'}
{attribute 'enable_dynamic_creation'}
FUNCTION_BLOCK FB_BACnet_AV_5P EXTENDS FB_BACnet_AV
VAR_INPUT
	bEnSfty					: BOOL;
	fValSfty				: REAL;
	bEnCrit					: BOOL;
	fValCrit				: REAL;
	bEnManLoc				: BOOL;
	fValManLoc				: REAL;
END_VAR
VAR_INPUT CONSTANT PERSISTENT
	{region 'Operational Parameters'}
		{attribute 'parameterCategory':='Manual'}
		bEnManualRm : BOOL;
		{attribute 'parameterCategory':='Manual'}
		fValManualRm : REAL;
	{endregion}
END_VAR

SUPER^();

METHOD PROTECTED OnObjectStateChanged
SUPER^.OnObjectStateChanged();

CASE (tState) OF
	TCOM_STATE.TCOM_STATE_PREOP:
		// SyncHandler:
		RequestSyncHandlers(1, 4);
		
	TCOM_STATE.TCOM_STATE_SAFEOP:
		SyncPropertyPvPrio(E_BACnetPropIdentifier.PropPresentValue, SIZEOF(fValSfty), ADR(fValSfty), ADR(bEnSfty), BACnet_Param.ePrio_LifeSafety, 0, eFullSync_InitPLC, TRUE);
		SyncPropertyPvPrio(E_BACnetPropIdentifier.PropPresentValue, SIZEOF(fValCrit), ADR(fValCrit), ADR(bEnCrit), BACnet_Param.ePrio_Critical, 0, eFullSync_InitPLC, TRUE);
		SyncPropertyPvPrio(E_BACnetPropIdentifier.PropPresentValue, SIZEOF(fValManLoc), ADR(fValManLoc), ADR(bEnManLoc), BACnet_Param.ePrio_ManLocal, 0, eFullSync_InitPLC, TRUE);
		SyncPropertyPvPrio(E_BACnetPropIdentifier.PropPresentValue, SIZEOF(fValManualRm), ADR(fValManualRm), ADR(bEnManualRm), BACnet_Param.ePrio_ManRemote, 0, eFullSync_InitPLC, TRUE);
		
	TCOM_STATE.TCOM_STATE_OP:
		;
	
END_CASE
END_METHOD

PROPERTY EnManualRm : BOOL
GET
EnManualRm := bEnManualRm;
END_GET
SET
bEnManualRm := EnManualRm;
END_SET
END_PROPERTY

PROPERTY ValManualRm : REAL
GET
ValManualRm := fValManualRm;
END_GET
SET
fValManualRm := ValManualRm;
END_SET
END_PROPERTY

END_FUNCTION_BLOCK

// POUs/Local/Objects/FB_BACnet_AV_Disp
// Analog Setpoint Object for Operation
// - Used to display a value
{attribute 'enable_dynamic_creation'}
FUNCTION_BLOCK FB_BACnet_AV_Disp EXTENDS FB_BACnet_Object
VAR_INPUT
	fVal			: REAL;
END_VAR
VAR_INPUT CONSTANT PERSISTENT
	{region 'Variable Parameters'}
		{attribute 'parameterCategory':='Value'}
		fCOVIncrement : REAL := 0.1;
		{attribute 'parameterCategory':='Value'}
		eUnit : E_BA_Unit := E_BA_Unit.eOther_NoUnits;
	{endregion}
END_VAR
VAR_OUTPUT
	fPresentValue	: REAL;
END_VAR

IF bReady THEN
	fPresentValue := fVal;
ELSE
	fPresentValue := 0;
END_IF

SUPER^();

METHOD PROTECTED OnObjectStateChanged
SUPER^.OnObjectStateChanged();

CASE (tState) OF
	TCOM_STATE.TCOM_STATE_PREOP:
		// SyncHandler:
		RequestSyncHandlers(0, 3);
		
		// Properties:
		// EnableProperty(E_BACnetPropIdentifier.PropDeviceType, FALSE);
		EnableProperty(E_BACnetPropIdentifier.PropNotificationClass, FALSE);
		EnableProperty(E_BACnetPropIdentifier.PropNotifyType, FALSE);
		EnableProperty(E_BACnetPropIdentifier.PropEventEnable, FALSE);
		EnableProperty(E_BACnetPropIdentifier.PropEventTimeStamps, FALSE);
		EnableProperty(E_BACnetPropIdentifier.PropEventMessageTexts, FALSE);
		EnableProperty(E_BACnetPropIdentifier.PropEventMessageTextsConfig, FALSE);
		EnableProperty(E_BACnetPropIdentifier.PropTimeDelay, FALSE);
		EnableProperty(E_BACnetPropIdentifier.PropAckedTransitions, FALSE);
		EnableProperty(E_BACnetPropIdentifier.PropReliability, FALSE);
		EnableProperty(E_BACnetPropIdentifier.PropEventDetectionEnable, FALSE);
		EnableProperty(E_BACnetPropIdentifier.PropEventAlgorithmInhibit, FALSE);
		EnableProperty(E_BACnetPropIdentifier.PropTimeDelayNormal, FALSE);
		EnableProperty(E_BACnetPropIdentifier.PropReliabilityEvaluationInhibit, FALSE);
		EnableProperty(E_BACnetPropIdentifier.PropLimitEnable, FALSE);
		EnableProperty(E_BACnetPropIdentifier.PropHighLimit, FALSE);
		EnableProperty(E_BACnetPropIdentifier.PropLowLimit, FALSE);
		EnableProperty(E_BACnetPropIdentifier.PropDeadband, FALSE);
		EnableProperty(E_BACnetPropIdentifier.PropRelinquishDefault, FALSE);
		EnableProperty(E_BACnetPropIdentifier.PropPriorityArray, FALSE);
		EnableProperty(E_BACnetPropIdentifier.PropCurrentlyActivePriority, FALSE);
		
		WriteProtectProperty(E_BACnetPropIdentifier.PropOutOfService, TRUE);
		// EnableProperty(E_BACnetPropIdentifier.PropStatusFlags, FALSE);
		// EnableProperty(E_BACnetPropIdentifier.PropEventState, FALSE);
		
		WriteProtectProperty(E_BACnetPropIdentifier.PropPresentValue, TRUE);
		
	TCOM_STATE.TCOM_STATE_SAFEOP:
		SyncProperty(E_BACnetPropIdentifier.PropPresentValue, SIZEOF(fVal), ADR(fVal), 0, eSync_ToSupplement, TRUE);
		
	TCOM_STATE.TCOM_STATE_OP:
		SyncProperty(E_BACnetPropIdentifier.PropUnits, SIZEOF(eUnit), ADR(eUnit), 0, eFullSync_InitPLC, FALSE);
		SyncProperty(E_BACnetPropIdentifier.PropCovIncrement, SIZEOF(fCOVIncrement), ADR(fCOVIncrement), 0, eFullSync_InitPLC, FALSE);
		
END_CASE
END_METHOD

METHOD FB_init : BOOL
VAR_INPUT
	bInitRetains : BOOL; // if TRUE, the retain variables are initialized (warm start / cold start)
	bInCopyCode : BOOL;  // if TRUE, the instance afterwards gets moved into the copy code (online change)
END_VAR
eObjectType := E_BACnetObjType.ObjAnalogValue;
END_METHOD

END_FUNCTION_BLOCK

// POUs/Local/Objects/FB_BACnet_AV_Setp
// Analog Setpoint Object for Operation
// - Used to define a setpoint by user
{attribute 'enable_dynamic_creation'}
FUNCTION_BLOCK FB_BACnet_AV_Setp EXTENDS FB_BACnet_Object
VAR_INPUT CONSTANT PERSISTENT
	{region 'Variable Parameters'}
		{attribute 'parameterCategory':='Value'}
		fCOVIncrement : REAL := 0.1;
		{attribute 'parameterCategory':='Value'}
		eUnit : E_BA_Unit := E_BA_Unit.eOther_NoUnits;
	{endregion}
	{region 'Operational Parameters'}
		{attribute 'parameterCategory':='Value'}
		fValue : REAL;
	{endregion}
END_VAR
VAR_OUTPUT
	fPresentValue	: REAL;
END_VAR

IF bReady THEN
	fPresentValue := fValue;
ELSE
	fPresentValue := 0;
END_IF

SUPER^();

METHOD PROTECTED OnObjectStateChanged
SUPER^.OnObjectStateChanged();

CASE (tState) OF
	TCOM_STATE.TCOM_STATE_PREOP:
		// SyncHandler:
		RequestSyncHandlers(0, 3);
		
		// Properties:
		// DisableProperty(E_BACnetPropIdentifier.PropDeviceType, FALSE);
		EnableProperty(E_BACnetPropIdentifier.PropNotificationClass, FALSE);
		EnableProperty(E_BACnetPropIdentifier.PropNotifyType, FALSE);
		EnableProperty(E_BACnetPropIdentifier.PropEventEnable, FALSE);
		EnableProperty(E_BACnetPropIdentifier.PropEventTimeStamps, FALSE);
		EnableProperty(E_BACnetPropIdentifier.PropEventMessageTexts, FALSE);
		EnableProperty(E_BACnetPropIdentifier.PropEventMessageTextsConfig, FALSE);
		EnableProperty(E_BACnetPropIdentifier.PropTimeDelay, FALSE);
		EnableProperty(E_BACnetPropIdentifier.PropAckedTransitions, FALSE);
		EnableProperty(E_BACnetPropIdentifier.PropReliability, FALSE);
		EnableProperty(E_BACnetPropIdentifier.PropEventDetectionEnable, FALSE);
		EnableProperty(E_BACnetPropIdentifier.PropEventAlgorithmInhibit, FALSE);
		EnableProperty(E_BACnetPropIdentifier.PropTimeDelayNormal, FALSE);
		EnableProperty(E_BACnetPropIdentifier.PropReliabilityEvaluationInhibit, FALSE);
		EnableProperty(E_BACnetPropIdentifier.PropLimitEnable, FALSE);
		EnableProperty(E_BACnetPropIdentifier.PropHighLimit, FALSE);
		EnableProperty(E_BACnetPropIdentifier.PropLowLimit, FALSE);
		EnableProperty(E_BACnetPropIdentifier.PropDeadband, FALSE);
		EnableProperty(E_BACnetPropIdentifier.PropRelinquishDefault, FALSE);
		EnableProperty(E_BACnetPropIdentifier.PropPriorityArray, FALSE);
		EnableProperty(E_BACnetPropIdentifier.PropCurrentlyActivePriority, FALSE);
		
		WriteProtectProperty(E_BACnetPropIdentifier.PropOutOfService, TRUE);
		// EnableProperty(E_BACnetPropIdentifier.PropStatusFlags, FALSE);
		// EnableProperty(E_BACnetPropIdentifier.PropEventState, FALSE);
		
	TCOM_STATE.TCOM_STATE_SAFEOP:
		;
		
	TCOM_STATE.TCOM_STATE_OP:
		SyncProperty(E_BACnetPropIdentifier.PropPresentValue, SIZEOF(fValue), ADR(fValue), 0, eFullSync_InitPLC, FALSE);
		
		SyncProperty(E_BACnetPropIdentifier.PropUnits, SIZEOF(eUnit), ADR(eUnit), 0, eFullSync_InitPLC, FALSE);
		SyncProperty(E_BACnetPropIdentifier.PropCovIncrement, SIZEOF(fCOVIncrement), ADR(fCOVIncrement), 0, eFullSync_InitPLC, FALSE);
END_CASE
END_METHOD

METHOD FB_init : BOOL
VAR_INPUT
	bInitRetains : BOOL; // if TRUE, the retain variables are initialized (warm start / cold start)
	bInCopyCode : BOOL;  // if TRUE, the instance afterwards gets moved into the copy code (online change)
END_VAR
eObjectType := E_BACnetObjType.ObjAnalogValue;
END_METHOD

END_FUNCTION_BLOCK

// POUs/Local/Objects/FB_BACnet_BI_Raw
// Binary Input Object
// - Raw communication
{attribute 'pin_presentation_order_outputs' := 'bPresentValue,bEvent,eReliability'}
{attribute 'enable_dynamic_creation'}
FUNCTION_BLOCK FB_BACnet_BI_Raw EXTENDS FB_BACnet_BaseBI
VAR_INPUT
	bRawValue					: BOOL;				// Raw value
END_VAR

SUPER^();

METHOD PROTECTED OnObjectStateChanged
SUPER^.OnObjectStateChanged();

CASE (tState) OF
	TCOM_STATE.TCOM_STATE_PREOP:
		// SyncHandler:
		RequestSyncHandlers(0, 1);

	TCOM_STATE.TCOM_STATE_SAFEOP:
		SyncProperty(E_BACnetPropIdentifier.PropRawIoBinaryValueBOOL, SIZEOF(bRawValue), ADR(bRawValue), 0, eSync_ToSupplement, TRUE);
		
	TCOM_STATE.TCOM_STATE_OP:
		;

END_CASE
END_METHOD

END_FUNCTION_BLOCK

// POUs/Local/Objects/[Base]/FB_BACnet_BaseBI
FUNCTION_BLOCK FB_BACnet_BaseBI EXTENDS FB_BACnet_EventObject
VAR_INPUT CONSTANT PERSISTENT
	{region 'Variable Parameters'}
		{attribute 'parameterCategory':='Value'}
		bOutOfService : BOOL;
		{attribute 'parameterCategory':='Value'}
		{attribute 'TcEncoding':='UTF-8'}
		sInactiveText : T_BACnet_StateText;
		{attribute 'parameterCategory':='Value'}
		{attribute 'TcEncoding':='UTF-8'}
		sActiveText : T_BACnet_StateText;
		
		{attribute 'parameterCategory':='Hardware'}
		{attribute 'TcEncoding':='UTF-8'}
		sDeviceType : STRING;
		
		{attribute 'parameterCategory':='EventConfig'}
		bAlarmValue : BOOL := TRUE;
		
		{attribute 'parameterCategory':='Config'}
		ePolarity : E_BA_Polarity := E_BA_Polarity.eNormal;
			 
		{attribute 'parameterCategory':='StateChange'}
		nChangeOfStateCount : UDINT;
		
		{attribute 'parameterCategory':='ActiveTime'}
		{attribute 'parameterUnit':= 's'}
		nElapsedActiveTime : UDINT;
	{endregion}
END_VAR
VAR_OUTPUT
	bPresentValue			: BOOL;
END_VAR
VAR
	{region 'Output-Properties'}
		{attribute 'parameterCategory':='StateChange'}
		stChangeOfStateTime : ST_BA_DateTime;
		{attribute 'parameterCategory':='StateChange'}
		stTimeOfStateCountReset : ST_BA_DateTime;
		
		{attribute 'parameterCategory':='ActiveTime'}
		stTimeOfActiveTimeReset : ST_BA_DateTime;
	{endregion}
END_VAR

SUPER^();

METHOD PROTECTED OnObjectStateChanged
SUPER^.OnObjectStateChanged();

CASE (tState) OF
	TCOM_STATE.TCOM_STATE_PREOP:
		// SyncHandler:
		RequestSyncHandlers(4, 8);
		
		// Properties:
		IF (BACnet_Param.bStateText_WriteProtect) THEN
			WriteProtectProperty(E_BACnetPropIdentifier.PropActiveText, TRUE);
			WriteProtectProperty(E_BACnetPropIdentifier.PropInactiveText, TRUE);
		END_IF
		
		// Ensure UTF-8 Encoding:
		F_BA_EnsureUTF8(ADR(sDeviceType), SIZEOF(sDeviceType));
		F_BA_EnsureUTF8(ADR(sInactiveText), SIZEOF(sInactiveText));
		F_BA_EnsureUTF8(ADR(sActiveText), SIZEOF(sActiveText));

	TCOM_STATE.TCOM_STATE_SAFEOP:
		SyncProperty(E_BACnetPropIdentifier.PropPresentValue, SIZEOF(bPresentValue), ADR(bPresentValue), 0, eSync_FromSupplement, TRUE);
		
	TCOM_STATE.TCOM_STATE_OP:
		SyncProperty(E_BACnetPropIdentifier.PropAlarmValue, SIZEOF(bAlarmValue), ADR(bAlarmValue), 0, eFullSync_InitPLC, FALSE);
		SyncProperty(E_BACnetPropIdentifier.PropOutOfService, SIZEOF(bOutOfService), ADR(bOutOfService), 0, eFullSync_InitPLC, FALSE);
		SyncProperty(E_BACnetPropIdentifier.PropActiveText, SIZEOF(sActiveText), ADR(sActiveText), 0, eFullSync_InitPLC, FALSE);	
		SyncProperty(E_BACnetPropIdentifier.PropInactiveText, SIZEOF(sInactiveText), ADR(sInactiveText), 0, eFullSync_InitPLC, FALSE);
		SyncProperty(E_BACnetPropIdentifier.PropPolarity, SIZEOF(ePolarity), ADR(ePolarity), 0, eFullSync_InitPLC, FALSE);
		SyncProperty(E_BACnetPropIdentifier.PropDeviceType, SIZEOF(sDeviceType), ADR(sDeviceType), 0, eFullSync_InitPLC, FALSE);

		SyncProperty(E_BACnetPropIdentifier.PropChangeOfStateCount, SIZEOF(nChangeOfStateCount), ADR(nChangeOfStateCount), 0, eFullSync_InitPLC, FALSE);
		SyncProperty(E_BACnetPropIdentifier.PropChangeOfStateTime, SIZEOF(stChangeOfStateTime), ADR(stChangeOfStateTime), 0, eSync_FromSupplement, FALSE);
		SyncProperty(E_BACnetPropIdentifier.PropTimeOfStateCountReset, SIZEOF(stTimeOfStateCountReset), ADR(stTimeOfStateCountReset), 0, eSync_FromSupplement, FALSE);

		SyncProperty(E_BACnetPropIdentifier.PropElapsedActiveTime, SIZEOF(nElapsedActiveTime), ADR(nElapsedActiveTime), 0, eFullSync_InitPLC, FALSE);
		SyncProperty(E_BACnetPropIdentifier.PropTimeOfActiveTimeReset, SIZEOF(stTimeOfActiveTimeReset), ADR(stTimeOfActiveTimeReset), 0, eSync_FromSupplement, FALSE);
		
END_CASE
END_METHOD

METHOD FB_init : BOOL
VAR_INPUT
	bInitRetains : BOOL; // if TRUE, the retain variables are initialized (warm start / cold start)
	bInCopyCode : BOOL;  // if TRUE, the instance afterwards gets moved into the copy code (online change)
END_VAR
eObjectType := E_BACnetObjType.ObjBinaryInput;
END_METHOD

PROPERTY ChangeOfStateTime : ST_BA_DateTime
GET
ChangeOfStateTime := stChangeOfStateTime;
END_GET
END_PROPERTY

PROPERTY TimeOfActiveTimeReset : ST_BA_DateTime
GET
TimeOfActiveTimeReset := stTimeOfActiveTimeReset;
END_GET
END_PROPERTY

PROPERTY TimeOfStateCountReset : ST_BA_DateTime
GET
TimeOfStateCountReset := stTimeOfStateCountReset;
END_GET
END_PROPERTY

END_FUNCTION_BLOCK

// POUs/Local/Objects/FB_BACnet_BO_Raw
// Binary Output Object
// - Raw communication
// - 1 Priority
{attribute 'pin_presentation_order_outputs' := 'fPresentValue,bEvent,eReliability'}
{attribute 'enable_dynamic_creation'}
FUNCTION_BLOCK FB_BACnet_BO_Raw EXTENDS FB_BACnet_BaseBO
VAR_INPUT
	bRawOverridden				: BOOL;				// Raw overridden

	bEnFeedback					: BOOL;				// Enable of writing to Feedback Value (optional)
	bRawValFeedback				: BOOL;				// Raw feedback Value
END_VAR
VAR_OUTPUT
	bRawValue					: BOOL;				// Raw value
END_VAR

IF (bReady) THEN
	// Feedback Value:
	_bFeedbackValue := SEL(bEnFeedback, bPresentValue, bRawValFeedback);
END_IF

SUPER^();

METHOD PROTECTED OnObjectStateChanged
SUPER^.OnObjectStateChanged();

CASE (tState) OF
	TCOM_STATE.TCOM_STATE_PREOP:
		// SyncHandler:
		RequestSyncHandlers(1, 1);

	TCOM_STATE.TCOM_STATE_SAFEOP:
		SyncProperty(E_BACnetPropIdentifier.PropRawIoBinaryValueBOOL, SIZEOF(bRawValue), ADR(bRawValue), 0, eSync_FromSupplement, TRUE);
		
	TCOM_STATE.TCOM_STATE_OP:
		SyncProperty(E_BACnetPropIdentifier.PropRawIoStateOverrideInverted, SIZEOF(bRawOverridden), ADR(bRawOverridden), 0, eSync_ToSupplement, FALSE);

END_CASE
END_METHOD

END_FUNCTION_BLOCK

// POUs/Local/Objects/[Base]/FB_BACnet_BaseBO
FUNCTION_BLOCK FB_BACnet_BaseBO EXTENDS FB_BACnet_EventObject
VAR_INPUT
	bEnPgm			: BOOL;
	bValPgm			: BOOL;
END_VAR
VAR_INPUT CONSTANT PERSISTENT
	{region 'Variable Parameters'}
		{attribute 'parameterCategory':='General'}
		{attribute 'parameterUnit':= 's'}
		nMinimumOffTime : UDINT;
		{attribute 'parameterCategory':='General'}
		{attribute 'parameterUnit':= 's'}
		nMinimumOnTime : UDINT;
		
		{attribute 'parameterCategory':='Value'}
		bRelinquishDefault : BOOL;
		{attribute 'parameterCategory':='Value'}
		bOutOfService : BOOL;
		{attribute 'parameterCategory':='Value'}
		{attribute 'TcEncoding':='UTF-8'}
		sInactiveText : T_BACnet_StateText;
		{attribute 'parameterCategory':='Value'}
		{attribute 'TcEncoding':='UTF-8'}
		sActiveText : T_BACnet_StateText;
		
		{attribute 'parameterCategory':='Hardware'}
		{attribute 'TcEncoding':='UTF-8'}
		sDeviceType : STRING;
		
		{attribute 'parameterCategory':='Config'}
		ePolarity : E_BA_Polarity := E_BA_Polarity.eNormal;
			 
		{attribute 'parameterCategory':='StateChange'}
		nChangeOfStateCount : UDINT;
		
		{attribute 'parameterCategory':='ActiveTime'}
		{attribute 'parameterUnit':= 's'}
		nElapsedActiveTime : UDINT;
	{endregion}
END_VAR
VAR_OUTPUT
	bPresentValue		: BOOL;
	eActivePrio			: E_BACnet_Priority;			// Indicates the currently active priority of the priority array
END_VAR
VAR
	{region 'Output-Properties'}
		{attribute 'parameterCategory':='StateChange'}
		stChangeOfStateTime : ST_BA_DateTime;
		{attribute 'parameterCategory':='StateChange'}
		stTimeOfStateCountReset : ST_BA_DateTime;
		
		{attribute 'parameterCategory':='ActiveTime'}
		stTimeOfActiveTimeReset : ST_BA_DateTime;
	{endregion}
END_VAR
VAR
	{region 'General'}
		_bFeedbackValue	: BOOL;
	{endregion}
END_VAR

SUPER^();

METHOD PROTECTED OnObjectStateChanged
SUPER^.OnObjectStateChanged();

CASE (tState) OF
	TCOM_STATE.TCOM_STATE_PREOP:
		// SyncHandler:
		RequestSyncHandlers(4, 12);
		
